// TIA Portal V20 export
FUNCTION_BLOCK "Sequence_1_MainPnP"   // FB246, LAD
AUTHOR : ERsystem_FA2_DH. Kim
// stored: IsIECCheckEnabled true, MemoryReserve 100, Namespace Unit1.Em5, SetENOAutomatically false
   VAR
      instSequenceLADStatus { ExternalWritable := 'False'} : "LAF_StatusLadSequence";
      instSequenceLADControl { ExternalWritable := 'False'} : "LAF_ControlLadSequence";
      statTonTime { ExternalWritable := 'False'} : Array[0..9999] of TON_TIME;
   END_VAR
   VAR_TEMP
      tempCustomerAction : Bool;   // Placeholder for possible actions
      tempDo_nothing_and_wait_for_init : Bool;   // Placeholder for doing nothing
      tempSafeStateCondition : Bool;   // Temp Condition for the equipment module to be in a safe state
   END_VAR
   VAR CONSTANT
      delayTime : Time := T#300ms;
      STEP_IDLE : DInt := 1;
      STEP_IMMEDIATE_STOP : DInt := 9001;   // Step executed when an immediate stop command is triggered for the sequence (i.e. when unit is in state aborting)
      JOB_10_STEP_01 : DInt := 1001;
      JOB_10_STEP_10 : DInt := 1010;
      JOB_10_STEP_11 : DInt := 1011;
      JOB_10_STEP_20 : DInt := 1020;
      JOB_10_STEP_21 : DInt := 1021;
      JOB_10_STEP_22 : DInt := 1022;
      JOB_10_STEP_30 : DInt := 1030;
      JOB_10_STEP_31 : DInt := 1031;
      JOB_10_STEP_40 : DInt := 1040;
      JOB_10_STEP_41 : DInt := 1041;
      JOB_10_STEP_50 : DInt := 1050;
      JOB_10_STEP_60 : DInt := 1060;
      JOB_10_STEP_70 : DInt := 1070;
      JOB_10_STEP_71 : DInt := 1071;
      JOB_10_STEP_80 : DInt := 1080;
      JOB_10_STEP_81 : DInt := 1081;
      JOB_10_STEP_90 : DInt := 1090;
      JOB_1_STEP_01 : DInt := 101;
      JOB_1_STEP_10 : DInt := 110;
      JOB_1_STEP_11 : DInt := 111;
      JOB_1_STEP_12 : DInt := 112;
      JOB_1_STEP_13 : DInt := 113;
      JOB_1_STEP_14 : DInt := 114;
      JOB_1_STEP_15 : DInt := 115;
      JOB_1_STEP_16 : DInt := 116;
      JOB_1_STEP_17 : DInt := 117;
      JOB_1_STEP_18 : DInt := 118;
      JOB_1_STEP_19 : DInt := 119;
      JOB_1_STEP_20 : DInt := 120;
      JOB_1_STEP_21 : DInt := 121;
      JOB_1_STEP_22 : DInt := 122;
      JOB_1_STEP_23 : DInt := 123;
      JOB_1_STEP_24 : DInt := 124;
      JOB_1_STEP_25 : DInt := 125;
      JOB_1_STEP_26 : DInt := 126;
      JOB_1_STEP_27 : DInt := 127;
      JOB_1_STEP_28 : DInt := 128;
      JOB_1_STEP_29 : DInt := 129;
      JOB_1_STEP_30 : DInt := 130;
      JOB_1_STEP_31 : DInt := 131;
      JOB_1_STEP_32 : DInt := 132;
      JOB_1_STEP_33 : DInt := 133;
      JOB_1_STEP_34 : DInt := 134;
      JOB_1_STEP_35 : DInt := 135;
      JOB_1_STEP_36 : DInt := 136;
      JOB_1_STEP_37 : DInt := 137;
      JOB_1_STEP_38 : DInt := 138;
      JOB_1_STEP_39 : DInt := 139;
      JOB_1_STEP_40 : DInt := 140;
      JOB_1_STEP_41 : DInt := 141;
      JOB_1_STEP_42 : DInt := 142;
      JOB_1_STEP_43 : DInt := 143;
      JOB_1_STEP_44 : DInt := 144;
      JOB_1_STEP_45 : DInt := 145;
      JOB_1_STEP_46 : DInt := 146;
      JOB_1_STEP_47 : DInt := 147;
      JOB_1_STEP_48 : DInt := 148;
      JOB_1_STEP_49 : DInt := 149;
      JOB_1_STEP_50 : DInt := 150;
      JOB_1_STEP_80 : DInt := 180;
      JOB_1_STEP_81 : DInt := 181;
      JOB_1_STEP_82 : DInt := 182;
      JOB_1_STEP_83 : DInt := 183;
      JOB_1_STEP_84 : DInt := 184;
      JOB_1_STEP_85 : DInt := 185;
      JOB_1_STEP_86 : DInt := 186;
      JOB_1_STEP_87 : DInt := 187;
      JOB_1_STEP_88 : DInt := 188;
      JOB_1_STEP_89 : DInt := 189;
      JOB_1_STEP_90 : DInt := 190;
      JOB_2_STEP_01 : DInt := 201;
      JOB_2_STEP_10 : DInt := 210;
      JOB_2_STEP_20 : DInt := 220;
      JOB_2_STEP_30 : DInt := 230;
      JOB_2_STEP_40 : DInt := 240;
      JOB_2_STEP_50 : DInt := 250;
      JOB_2_STEP_60 : DInt := 260;
      JOB_2_STEP_80 : DInt := 280;
      JOB_2_STEP_90 : DInt := 290;
      JOB_3_STEP_01 : DInt := 301;
      JOB_3_STEP_10 : DInt := 310;
      JOB_3_STEP_20 : DInt := 320;
      JOB_3_STEP_30 : DInt := 330;
      JOB_3_STEP_40 : DInt := 340;
      JOB_3_STEP_50 : DInt := 350;
      JOB_3_STEP_60 : DInt := 360;
      JOB_3_STEP_80 : DInt := 380;
      JOB_3_STEP_90 : DInt := 390;
      JOB_4_STEP_01 : DInt := 401;
      JOB_4_STEP_20 : DInt := 420;
      JOB_4_STEP_30 : DInt := 430;
      JOB_4_STEP_90 : DInt := 490;
      JOB_5_STEP_01 : DInt := 501;
      JOB_5_STEP_20 : DInt := 520;
      JOB_5_STEP_30 : DInt := 530;
      JOB_5_STEP_40 : DInt := 540;
      JOB_5_STEP_50 : DInt := 550;
      JOB_5_STEP_60 : DInt := 560;
      JOB_5_STEP_80 : DInt := 580;
      JOB_5_STEP_90 : DInt := 590;
      JOB_6_STEP_01 : DInt := 601;
      JOB_6_STEP_10 : DInt := 610;
      JOB_6_STEP_20 : DInt := 620;
      JOB_6_STEP_30 : DInt := 630;
      JOB_6_STEP_40 : DInt := 640;
      JOB_6_STEP_50 : DInt := 650;
      JOB_6_STEP_60 : DInt := 660;
      JOB_6_STEP_80 : DInt := 680;
      JOB_6_STEP_90 : DInt := 690;
      FALSE : Bool := FALSE;
      TRUE : Bool := TRUE;
      kim_bool : Bool := true;
   END_VAR
   VAR_TEMP   // added for the SCL form of the ladder/FBD networks
      _w1 : Bool;
   END_VAR
BEGIN

REGION Network 1: BLOCK INFO HEADER
   // (company) / (C) Copyright (year)
   // ---------------------------------------------------------------------------------
   // Title:                             (Title of this block)
   // Comment/Function: (that is implemented in the block)
   // Library/Family:           (that the source is dedicated to)
   // Author:                        (department / person in charge / contact)
   // Target System:          (test system with FW version)
   // Engineering:              TIA Portal (SW version)
   // Restrictions:               (OB types, etc.)
   // Requirements:           (hardware, technological package, etc.)
   // ---------------------------------------------------------------------------------
   // Change log table:
   // Version          | Date             | Signature      | Expert in charge  | Changes applied ------------------------|----------------------|-------------------------|--------------------------------|-----------------------
   // 001.000.000 | yyyy-mm-dd | 0x00000000 | (name of expert) | First released version
END_REGION

REGION Network 2: DESCRIPTION
   // This is a template block provided by the Automation Framework. It can be used to create an own project.
   // The Block Info Header is prepared to put in your own data.
   // Description of the block could be added here and the docu created by Code2Docu.
END_REGION

REGION Network 3: ********************* CONTROL *************************
END_REGION

REGION Network 4: Sequence Control
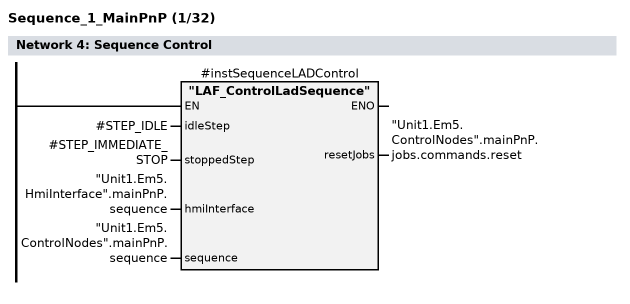
   RUNG wire#powerrail
      #instSequenceLADControl(idleStep := #STEP_IDLE, stoppedStep := #STEP_IMMEDIATE_STOP, hmiInterface := "Unit1.Em5.HmiInterface".mainPnP.sequence, sequence := "Unit1.Em5.ControlNodes".mainPnP.sequence, resetJobs => "Unit1.Em5.ControlNodes".mainPnP.jobs.commands.reset)
   END_RUNG
   // the same network as SCL:
   #instSequenceLADControl(idleStep := #STEP_IDLE,   // "LAF_ControlLadSequence"
                           stoppedStep := #STEP_IMMEDIATE_STOP,
                           hmiInterface := "Unit1.Em5.HmiInterface".mainPnP.sequence,
                           sequence := "Unit1.Em5.ControlNodes".mainPnP.sequence,
                           resetJobs => "Unit1.Em5.ControlNodes".mainPnP.jobs.commands.reset);
END_REGION

REGION Network 5: *************** JOB SELECT **************************
END_REGION

REGION Network 6: STEP IDLE
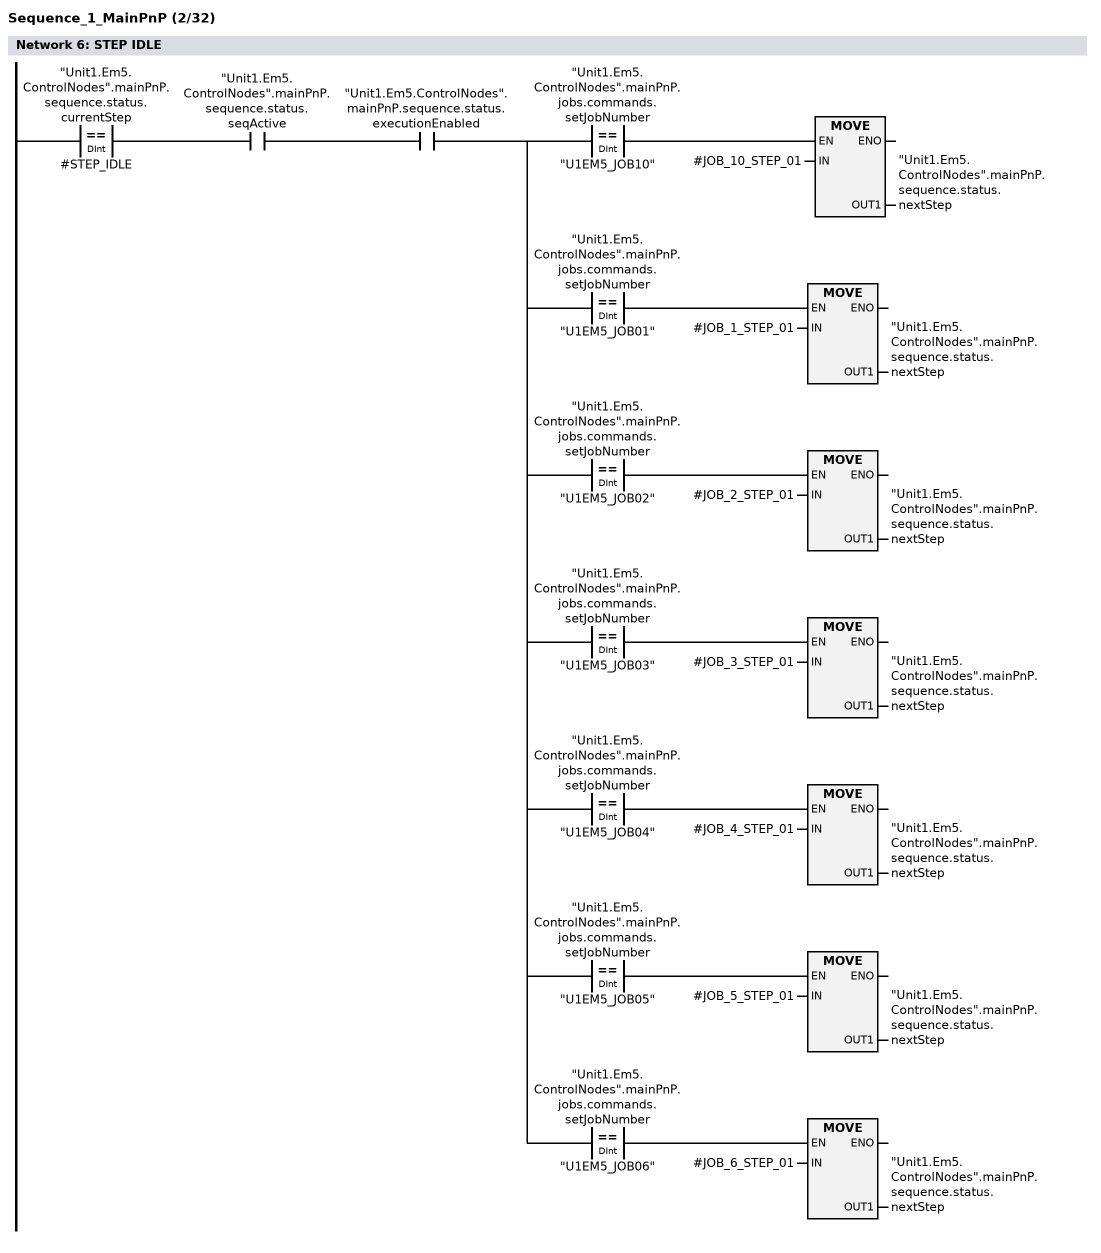
   RUNG wire#powerrail
      { S7_Templates := "SrcType := DInt" } EQ_Contact(in1 := "Unit1.Em5.ControlNodes".mainPnP.sequence.status.currentStep, in2 := #STEP_IDLE)
      Contact( "Unit1.Em5.ControlNodes".mainPnP.sequence.status.seqActive )
      Contact( "Unit1.Em5.ControlNodes".mainPnP.sequence.status.executionEnabled )
      wire#w1
      { S7_Templates := "SrcType := DInt" } EQ_Contact(in1 := "Unit1.Em5.ControlNodes".mainPnP.jobs.commands.setJobNumber, in2 := "U1EM5_JOB10")
      Move(in := #JOB_10_STEP_01, out1 => "Unit1.Em5.ControlNodes".mainPnP.sequence.status.nextStep)
   END_RUNG
   RUNG wire#w1
      { S7_Templates := "SrcType := DInt" } EQ_Contact(in1 := "Unit1.Em5.ControlNodes".mainPnP.jobs.commands.setJobNumber, in2 := "U1EM5_JOB01")
      Move(in := #JOB_1_STEP_01, out1 => "Unit1.Em5.ControlNodes".mainPnP.sequence.status.nextStep)
   END_RUNG
   RUNG wire#w1
      { S7_Templates := "SrcType := DInt" } EQ_Contact(in1 := "Unit1.Em5.ControlNodes".mainPnP.jobs.commands.setJobNumber, in2 := "U1EM5_JOB02")
      Move(in := #JOB_2_STEP_01, out1 => "Unit1.Em5.ControlNodes".mainPnP.sequence.status.nextStep)
   END_RUNG
   RUNG wire#w1
      { S7_Templates := "SrcType := DInt" } EQ_Contact(in1 := "Unit1.Em5.ControlNodes".mainPnP.jobs.commands.setJobNumber, in2 := "U1EM5_JOB03")
      Move(in := #JOB_3_STEP_01, out1 => "Unit1.Em5.ControlNodes".mainPnP.sequence.status.nextStep)
   END_RUNG
   RUNG wire#w1
      { S7_Templates := "SrcType := DInt" } EQ_Contact(in1 := "Unit1.Em5.ControlNodes".mainPnP.jobs.commands.setJobNumber, in2 := "U1EM5_JOB04")
      Move(in := #JOB_4_STEP_01, out1 => "Unit1.Em5.ControlNodes".mainPnP.sequence.status.nextStep)
   END_RUNG
   RUNG wire#w1
      { S7_Templates := "SrcType := DInt" } EQ_Contact(in1 := "Unit1.Em5.ControlNodes".mainPnP.jobs.commands.setJobNumber, in2 := "U1EM5_JOB05")
      Move(in := #JOB_5_STEP_01, out1 => "Unit1.Em5.ControlNodes".mainPnP.sequence.status.nextStep)
   END_RUNG
   RUNG wire#w1
      { S7_Templates := "SrcType := DInt" } EQ_Contact(in1 := "Unit1.Em5.ControlNodes".mainPnP.jobs.commands.setJobNumber, in2 := "U1EM5_JOB06")
      Move(in := #JOB_6_STEP_01, out1 => "Unit1.Em5.ControlNodes".mainPnP.sequence.status.nextStep)
   END_RUNG
   // the same network as SCL:
   #_w1 := ("Unit1.Em5.ControlNodes".mainPnP.sequence.status.currentStep = #STEP_IDLE) AND "Unit1.Em5.ControlNodes".mainPnP.sequence.status.seqActive AND "Unit1.Em5.ControlNodes".mainPnP.sequence.status.executionEnabled;
   IF #_w1 AND ("Unit1.Em5.ControlNodes".mainPnP.jobs.commands.setJobNumber = "U1EM5_JOB10") THEN
       "Unit1.Em5.ControlNodes".mainPnP.sequence.status.nextStep := #JOB_10_STEP_01;
   END_IF;
   IF #_w1 AND ("Unit1.Em5.ControlNodes".mainPnP.jobs.commands.setJobNumber = "U1EM5_JOB01") THEN
       "Unit1.Em5.ControlNodes".mainPnP.sequence.status.nextStep := #JOB_1_STEP_01;
   END_IF;
   IF #_w1 AND ("Unit1.Em5.ControlNodes".mainPnP.jobs.commands.setJobNumber = "U1EM5_JOB02") THEN
       "Unit1.Em5.ControlNodes".mainPnP.sequence.status.nextStep := #JOB_2_STEP_01;
   END_IF;
   IF #_w1 AND ("Unit1.Em5.ControlNodes".mainPnP.jobs.commands.setJobNumber = "U1EM5_JOB03") THEN
       "Unit1.Em5.ControlNodes".mainPnP.sequence.status.nextStep := #JOB_3_STEP_01;
   END_IF;
   IF #_w1 AND ("Unit1.Em5.ControlNodes".mainPnP.jobs.commands.setJobNumber = "U1EM5_JOB04") THEN
       "Unit1.Em5.ControlNodes".mainPnP.sequence.status.nextStep := #JOB_4_STEP_01;
   END_IF;
   IF #_w1 AND ("Unit1.Em5.ControlNodes".mainPnP.jobs.commands.setJobNumber = "U1EM5_JOB05") THEN
       "Unit1.Em5.ControlNodes".mainPnP.sequence.status.nextStep := #JOB_5_STEP_01;
   END_IF;
   IF #_w1 AND ("Unit1.Em5.ControlNodes".mainPnP.jobs.commands.setJobNumber = "U1EM5_JOB06") THEN
       "Unit1.Em5.ControlNodes".mainPnP.sequence.status.nextStep := #JOB_6_STEP_01;
   END_IF;
END_REGION

REGION Network 7: *************** JOB[10] EM HOMING ************************
END_REGION

REGION Network 8: Step[1001] : JOB[10] Condition
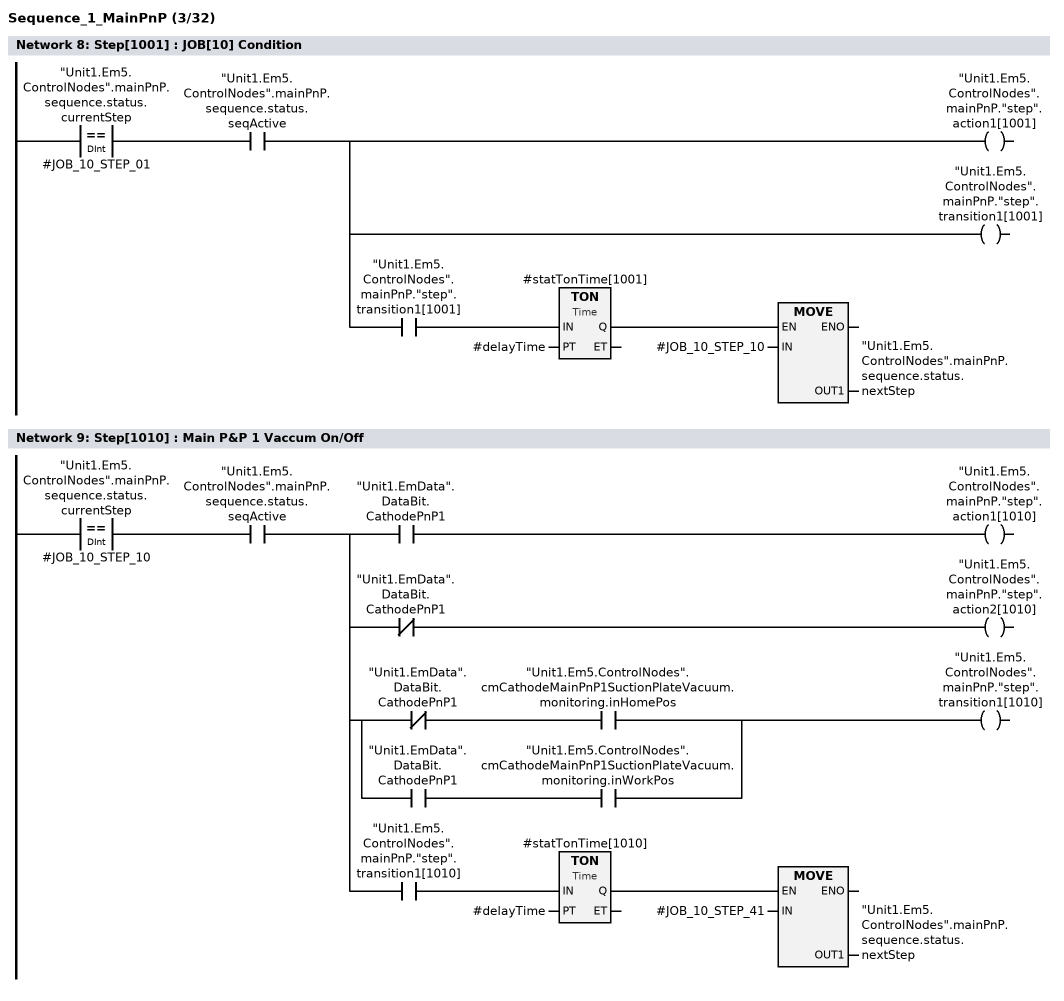
   RUNG wire#powerrail
      { S7_Templates := "SrcType := DInt" } EQ_Contact(in1 := "Unit1.Em5.ControlNodes".mainPnP.sequence.status.currentStep, in2 := #JOB_10_STEP_01)
      Contact( "Unit1.Em5.ControlNodes".mainPnP.sequence.status.seqActive )
      wire#w1
      Coil( "Unit1.Em5.ControlNodes".mainPnP."step".action1[1001] )
   END_RUNG
   RUNG wire#w1
      Coil( "Unit1.Em5.ControlNodes".mainPnP."step".transition1[1001] )
   END_RUNG
   RUNG wire#w1
      Contact( "Unit1.Em5.ControlNodes".mainPnP."step".transition1[1001] )
      { S7_Templates := "time_type := Time" } #statTonTime[1001].TON(pt := #delayTime, et =>)
      Move(in := #JOB_10_STEP_10, out1 => "Unit1.Em5.ControlNodes".mainPnP.sequence.status.nextStep)
   END_RUNG
   // the same network as SCL:
   "Unit1.Em5.ControlNodes".mainPnP."step".action1[1001] := ("Unit1.Em5.ControlNodes".mainPnP.sequence.status.currentStep = #JOB_10_STEP_01) AND "Unit1.Em5.ControlNodes".mainPnP.sequence.status.seqActive;
   "Unit1.Em5.ControlNodes".mainPnP."step".transition1[1001] := ("Unit1.Em5.ControlNodes".mainPnP.sequence.status.currentStep = #JOB_10_STEP_01) AND "Unit1.Em5.ControlNodes".mainPnP.sequence.status.seqActive;
   #statTonTime[1001].TON(IN := ("Unit1.Em5.ControlNodes".mainPnP.sequence.status.currentStep = #JOB_10_STEP_01) AND "Unit1.Em5.ControlNodes".mainPnP.sequence.status.seqActive AND "Unit1.Em5.ControlNodes".mainPnP."step".transition1[1001],
                          PT := #delayTime);
   IF #statTonTime[1001].Q THEN
       "Unit1.Em5.ControlNodes".mainPnP.sequence.status.nextStep := #JOB_10_STEP_10;
   END_IF;
END_REGION

REGION Network 9: Step[1010] : Main P&P 1 Vaccum On/Off
   RUNG wire#powerrail
      { S7_Templates := "SrcType := DInt" } EQ_Contact(in1 := "Unit1.Em5.ControlNodes".mainPnP.sequence.status.currentStep, in2 := #JOB_10_STEP_10)
      Contact( "Unit1.Em5.ControlNodes".mainPnP.sequence.status.seqActive )
      wire#w1
      Contact( "Unit1.EmData".DataBit.CathodePnP1 )
      Coil( "Unit1.Em5.ControlNodes".mainPnP."step".action1[1010] )
   END_RUNG
   RUNG wire#w1
      I_Contact( "Unit1.EmData".DataBit.CathodePnP1 )
      Coil( "Unit1.Em5.ControlNodes".mainPnP."step".action2[1010] )
   END_RUNG
   RUNG wire#w1
      I_Contact( "Unit1.EmData".DataBit.CathodePnP1 )
      Contact( "Unit1.Em5.ControlNodes".cmCathodeMainPnP1SuctionPlateVacuum.monitoring.inHomePos )
      wire#w2
      Coil( "Unit1.Em5.ControlNodes".mainPnP."step".transition1[1010] )
   END_RUNG
   RUNG wire#w1
      Contact( "Unit1.EmData".DataBit.CathodePnP1 )
      Contact( "Unit1.Em5.ControlNodes".cmCathodeMainPnP1SuctionPlateVacuum.monitoring.inWorkPos )
   END_RUNG wire#w2
   RUNG wire#w1
      Contact( "Unit1.Em5.ControlNodes".mainPnP."step".transition1[1010] )
      { S7_Templates := "time_type := Time" } #statTonTime[1010].TON(pt := #delayTime, et =>)
      Move(in := #JOB_10_STEP_41, out1 => "Unit1.Em5.ControlNodes".mainPnP.sequence.status.nextStep)
   END_RUNG
   // the same network as SCL:
   #_w1 := ("Unit1.Em5.ControlNodes".mainPnP.sequence.status.currentStep = #JOB_10_STEP_10) AND "Unit1.Em5.ControlNodes".mainPnP.sequence.status.seqActive;
   "Unit1.Em5.ControlNodes".mainPnP."step".action1[1010] := #_w1 AND "Unit1.EmData".DataBit.CathodePnP1;
   "Unit1.Em5.ControlNodes".mainPnP."step".action2[1010] := #_w1 AND NOT "Unit1.EmData".DataBit.CathodePnP1;
   "Unit1.Em5.ControlNodes".mainPnP."step".transition1[1010] := #_w1 AND ((NOT "Unit1.EmData".DataBit.CathodePnP1 AND "Unit1.Em5.ControlNodes".cmCathodeMainPnP1SuctionPlateVacuum.monitoring.inHomePos) OR ("Unit1.EmData".DataBit.CathodePnP1 AND "Unit1.Em5.ControlNodes".cmCathodeMainPnP1SuctionPlateVacuum.monitoring.inWorkPos));
   #statTonTime[1010].TON(IN := #_w1 AND "Unit1.Em5.ControlNodes".mainPnP."step".transition1[1010],
                          PT := #delayTime);
   IF #statTonTime[1010].Q THEN
       "Unit1.Em5.ControlNodes".mainPnP.sequence.status.nextStep := #JOB_10_STEP_41;
   END_IF;
END_REGION

REGION Network 10: Step[1041] : Main P&P 2 Vaccum On/Off
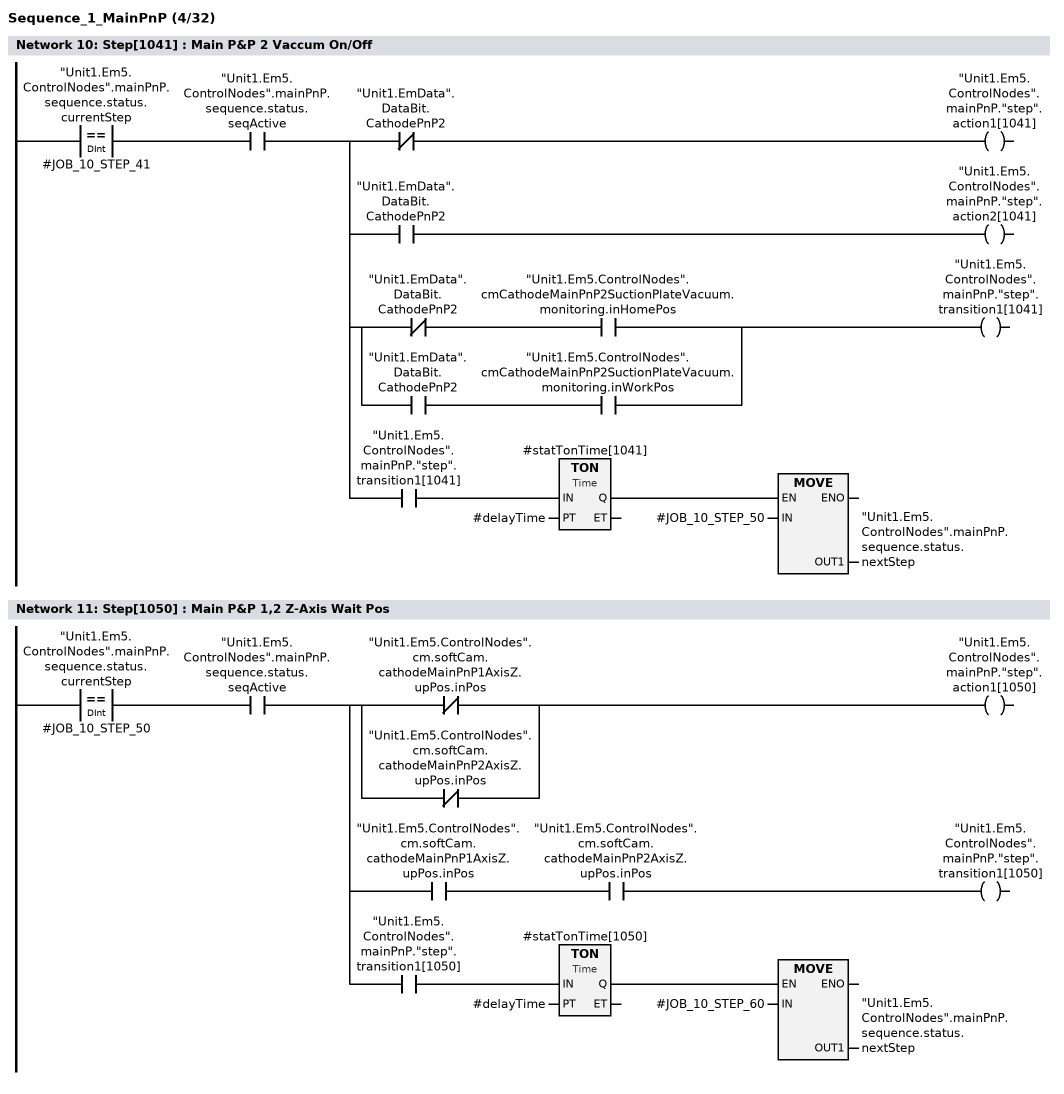
   RUNG wire#powerrail
      { S7_Templates := "SrcType := DInt" } EQ_Contact(in1 := "Unit1.Em5.ControlNodes".mainPnP.sequence.status.currentStep, in2 := #JOB_10_STEP_41)
      Contact( "Unit1.Em5.ControlNodes".mainPnP.sequence.status.seqActive )
      wire#w1
      I_Contact( "Unit1.EmData".DataBit.CathodePnP2 )
      Coil( "Unit1.Em5.ControlNodes".mainPnP."step".action1[1041] )
   END_RUNG
   RUNG wire#w1
      Contact( "Unit1.EmData".DataBit.CathodePnP2 )
      Coil( "Unit1.Em5.ControlNodes".mainPnP."step".action2[1041] )
   END_RUNG
   RUNG wire#w1
      I_Contact( "Unit1.EmData".DataBit.CathodePnP2 )
      Contact( "Unit1.Em5.ControlNodes".cmCathodeMainPnP2SuctionPlateVacuum.monitoring.inHomePos )
      wire#w2
      Coil( "Unit1.Em5.ControlNodes".mainPnP."step".transition1[1041] )
   END_RUNG
   RUNG wire#w1
      Contact( "Unit1.EmData".DataBit.CathodePnP2 )
      Contact( "Unit1.Em5.ControlNodes".cmCathodeMainPnP2SuctionPlateVacuum.monitoring.inWorkPos )
   END_RUNG wire#w2
   RUNG wire#w1
      Contact( "Unit1.Em5.ControlNodes".mainPnP."step".transition1[1041] )
      { S7_Templates := "time_type := Time" } #statTonTime[1041].TON(pt := #delayTime, et =>)
      Move(in := #JOB_10_STEP_50, out1 => "Unit1.Em5.ControlNodes".mainPnP.sequence.status.nextStep)
   END_RUNG
   // the same network as SCL:
   #_w1 := ("Unit1.Em5.ControlNodes".mainPnP.sequence.status.currentStep = #JOB_10_STEP_41) AND "Unit1.Em5.ControlNodes".mainPnP.sequence.status.seqActive;
   "Unit1.Em5.ControlNodes".mainPnP."step".action1[1041] := #_w1 AND NOT "Unit1.EmData".DataBit.CathodePnP2;
   "Unit1.Em5.ControlNodes".mainPnP."step".action2[1041] := #_w1 AND "Unit1.EmData".DataBit.CathodePnP2;
   "Unit1.Em5.ControlNodes".mainPnP."step".transition1[1041] := #_w1 AND ((NOT "Unit1.EmData".DataBit.CathodePnP2 AND "Unit1.Em5.ControlNodes".cmCathodeMainPnP2SuctionPlateVacuum.monitoring.inHomePos) OR ("Unit1.EmData".DataBit.CathodePnP2 AND "Unit1.Em5.ControlNodes".cmCathodeMainPnP2SuctionPlateVacuum.monitoring.inWorkPos));
   #statTonTime[1041].TON(IN := #_w1 AND "Unit1.Em5.ControlNodes".mainPnP."step".transition1[1041],
                          PT := #delayTime);
   IF #statTonTime[1041].Q THEN
       "Unit1.Em5.ControlNodes".mainPnP.sequence.status.nextStep := #JOB_10_STEP_50;
   END_IF;
END_REGION

REGION Network 11: Step[1050] : Main P&P 1,2 Z-Axis Wait Pos
   RUNG wire#powerrail
      { S7_Templates := "SrcType := DInt" } EQ_Contact(in1 := "Unit1.Em5.ControlNodes".mainPnP.sequence.status.currentStep, in2 := #JOB_10_STEP_50)
      Contact( "Unit1.Em5.ControlNodes".mainPnP.sequence.status.seqActive )
      wire#w1
      I_Contact( "Unit1.Em5.ControlNodes".cm.softCam.cathodeMainPnP1AxisZ.upPos.inPos )
      wire#w2
      Coil( "Unit1.Em5.ControlNodes".mainPnP."step".action1[1050] )
   END_RUNG
   RUNG wire#w1
      I_Contact( "Unit1.Em5.ControlNodes".cm.softCam.cathodeMainPnP2AxisZ.upPos.inPos )
   END_RUNG wire#w2
   RUNG wire#w1
      Contact( "Unit1.Em5.ControlNodes".cm.softCam.cathodeMainPnP1AxisZ.upPos.inPos )
      Contact( "Unit1.Em5.ControlNodes".cm.softCam.cathodeMainPnP2AxisZ.upPos.inPos )
      Coil( "Unit1.Em5.ControlNodes".mainPnP."step".transition1[1050] )
   END_RUNG
   RUNG wire#w1
      Contact( "Unit1.Em5.ControlNodes".mainPnP."step".transition1[1050] )
      { S7_Templates := "time_type := Time" } #statTonTime[1050].TON(pt := #delayTime, et =>)
      Move(in := #JOB_10_STEP_60, out1 => "Unit1.Em5.ControlNodes".mainPnP.sequence.status.nextStep)
   END_RUNG
   // the same network as SCL:
   #_w1 := ("Unit1.Em5.ControlNodes".mainPnP.sequence.status.currentStep = #JOB_10_STEP_50) AND "Unit1.Em5.ControlNodes".mainPnP.sequence.status.seqActive;
   "Unit1.Em5.ControlNodes".mainPnP."step".action1[1050] := #_w1 AND (NOT "Unit1.Em5.ControlNodes".cm.softCam.cathodeMainPnP1AxisZ.upPos.inPos OR NOT "Unit1.Em5.ControlNodes".cm.softCam.cathodeMainPnP2AxisZ.upPos.inPos);
   "Unit1.Em5.ControlNodes".mainPnP."step".transition1[1050] := #_w1 AND "Unit1.Em5.ControlNodes".cm.softCam.cathodeMainPnP1AxisZ.upPos.inPos AND "Unit1.Em5.ControlNodes".cm.softCam.cathodeMainPnP2AxisZ.upPos.inPos;
   #statTonTime[1050].TON(IN := #_w1 AND "Unit1.Em5.ControlNodes".mainPnP."step".transition1[1050],
                          PT := #delayTime);
   IF #statTonTime[1050].Q THEN
       "Unit1.Em5.ControlNodes".mainPnP.sequence.status.nextStep := #JOB_10_STEP_60;
   END_IF;
END_REGION

REGION Network 12: Step[1060] : Main P&P 1 Y-Axis Wait Pos
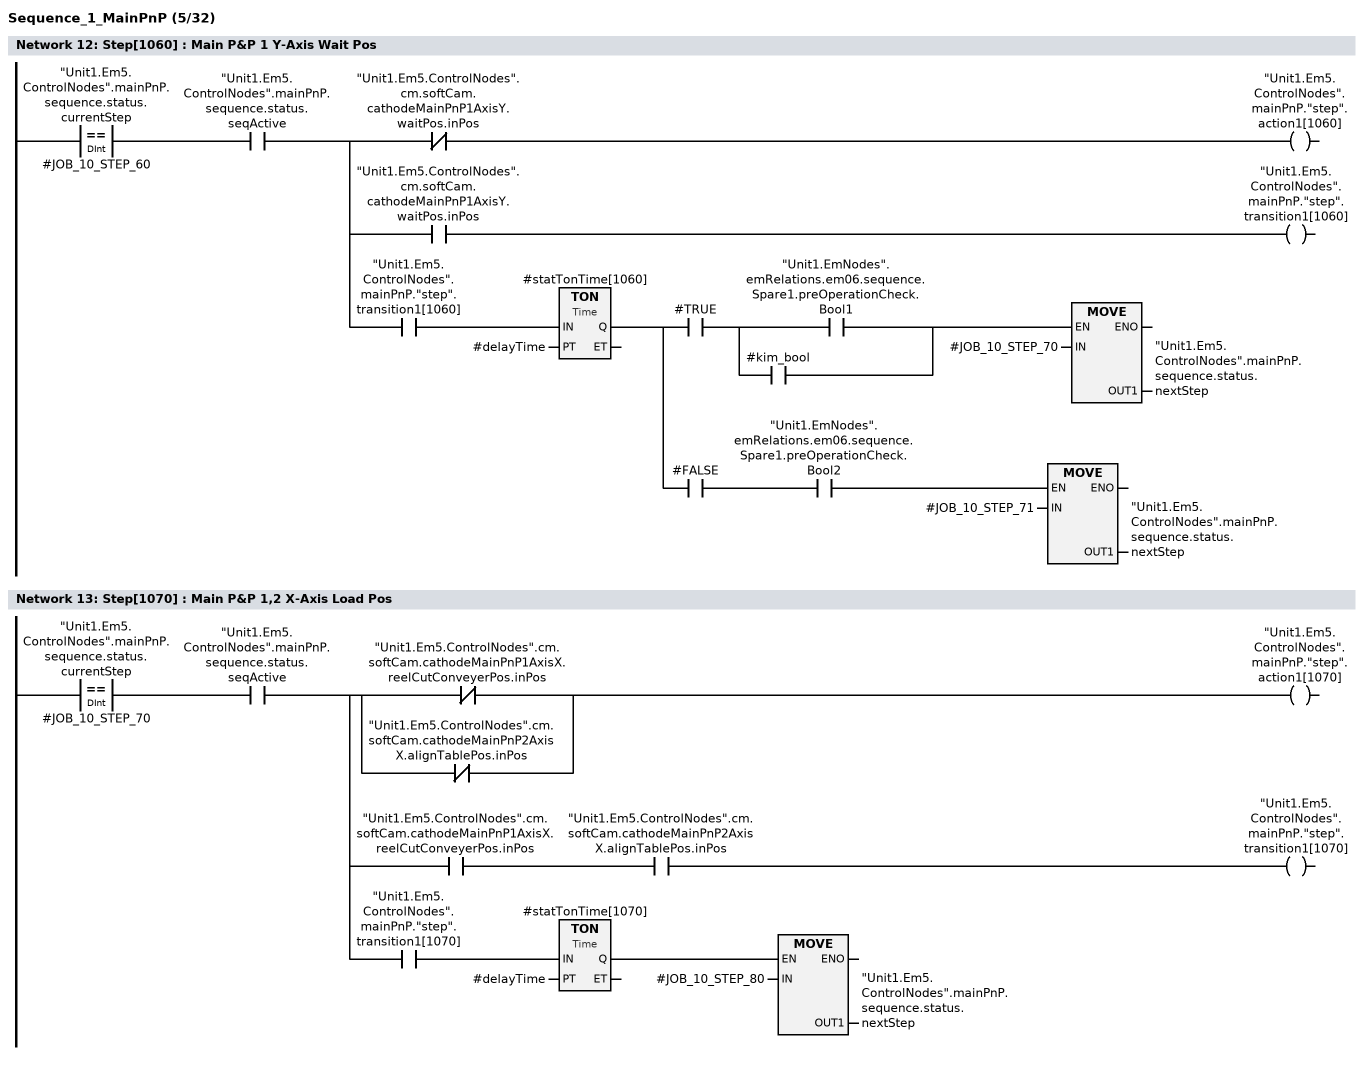
   RUNG wire#powerrail
      { S7_Templates := "SrcType := DInt" } EQ_Contact(in1 := "Unit1.Em5.ControlNodes".mainPnP.sequence.status.currentStep, in2 := #JOB_10_STEP_60)
      Contact( "Unit1.Em5.ControlNodes".mainPnP.sequence.status.seqActive )
      wire#w1
      I_Contact( "Unit1.Em5.ControlNodes".cm.softCam.cathodeMainPnP1AxisY.waitPos.inPos )
      Coil( "Unit1.Em5.ControlNodes".mainPnP."step".action1[1060] )
   END_RUNG
   RUNG wire#w1
      Contact( "Unit1.Em5.ControlNodes".cm.softCam.cathodeMainPnP1AxisY.waitPos.inPos )
      Coil( "Unit1.Em5.ControlNodes".mainPnP."step".transition1[1060] )
   END_RUNG
   RUNG wire#w1
      Contact( "Unit1.Em5.ControlNodes".mainPnP."step".transition1[1060] )
      { S7_Templates := "time_type := Time" } #statTonTime[1060].TON(pt := #delayTime, et =>)
      wire#w2
      Contact( #TRUE )
      wire#w3
      Contact( "Unit1.EmNodes".emRelations.em06.sequence.Spare1.preOperationCheck.Bool1 )
      wire#w4
      Move(in := #JOB_10_STEP_70, out1 => "Unit1.Em5.ControlNodes".mainPnP.sequence.status.nextStep)
   END_RUNG
   RUNG wire#w3
      Contact( #kim_bool )
   END_RUNG wire#w4
   RUNG wire#w2
      Contact( #FALSE )
      Contact( "Unit1.EmNodes".emRelations.em06.sequence.Spare1.preOperationCheck.Bool2 )
      Move(in := #JOB_10_STEP_71, out1 => "Unit1.Em5.ControlNodes".mainPnP.sequence.status.nextStep)
   END_RUNG
   // the same network as SCL:
   #_w1 := ("Unit1.Em5.ControlNodes".mainPnP.sequence.status.currentStep = #JOB_10_STEP_60) AND "Unit1.Em5.ControlNodes".mainPnP.sequence.status.seqActive;
   "Unit1.Em5.ControlNodes".mainPnP."step".action1[1060] := #_w1 AND NOT "Unit1.Em5.ControlNodes".cm.softCam.cathodeMainPnP1AxisY.waitPos.inPos;
   "Unit1.Em5.ControlNodes".mainPnP."step".transition1[1060] := #_w1 AND "Unit1.Em5.ControlNodes".cm.softCam.cathodeMainPnP1AxisY.waitPos.inPos;
   #statTonTime[1060].TON(IN := #_w1 AND "Unit1.Em5.ControlNodes".mainPnP."step".transition1[1060],
                          PT := #delayTime);
   IF #statTonTime[1060].Q AND #TRUE AND ("Unit1.EmNodes".emRelations.em06.sequence.Spare1.preOperationCheck.Bool1 OR #kim_bool) THEN
       "Unit1.Em5.ControlNodes".mainPnP.sequence.status.nextStep := #JOB_10_STEP_70;
   END_IF;
   IF #statTonTime[1060].Q AND #FALSE AND "Unit1.EmNodes".emRelations.em06.sequence.Spare1.preOperationCheck.Bool2 THEN
       "Unit1.Em5.ControlNodes".mainPnP.sequence.status.nextStep := #JOB_10_STEP_71;
   END_IF;
END_REGION

REGION Network 13: Step[1070] : Main P&P 1,2 X-Axis Load Pos
   RUNG wire#powerrail
      { S7_Templates := "SrcType := DInt" } EQ_Contact(in1 := "Unit1.Em5.ControlNodes".mainPnP.sequence.status.currentStep, in2 := #JOB_10_STEP_70)
      Contact( "Unit1.Em5.ControlNodes".mainPnP.sequence.status.seqActive )
      wire#w1
      I_Contact( "Unit1.Em5.ControlNodes".cm.softCam.cathodeMainPnP1AxisX.reelCutConveyerPos.inPos )
      wire#w2
      Coil( "Unit1.Em5.ControlNodes".mainPnP."step".action1[1070] )
   END_RUNG
   RUNG wire#w1
      I_Contact( "Unit1.Em5.ControlNodes".cm.softCam.cathodeMainPnP2AxisX.alignTablePos.inPos )
   END_RUNG wire#w2
   RUNG wire#w1
      Contact( "Unit1.Em5.ControlNodes".cm.softCam.cathodeMainPnP1AxisX.reelCutConveyerPos.inPos )
      Contact( "Unit1.Em5.ControlNodes".cm.softCam.cathodeMainPnP2AxisX.alignTablePos.inPos )
      Coil( "Unit1.Em5.ControlNodes".mainPnP."step".transition1[1070] )
   END_RUNG
   RUNG wire#w1
      Contact( "Unit1.Em5.ControlNodes".mainPnP."step".transition1[1070] )
      { S7_Templates := "time_type := Time" } #statTonTime[1070].TON(pt := #delayTime, et =>)
      Move(in := #JOB_10_STEP_80, out1 => "Unit1.Em5.ControlNodes".mainPnP.sequence.status.nextStep)
   END_RUNG
   // the same network as SCL:
   #_w1 := ("Unit1.Em5.ControlNodes".mainPnP.sequence.status.currentStep = #JOB_10_STEP_70) AND "Unit1.Em5.ControlNodes".mainPnP.sequence.status.seqActive;
   "Unit1.Em5.ControlNodes".mainPnP."step".action1[1070] := #_w1 AND (NOT "Unit1.Em5.ControlNodes".cm.softCam.cathodeMainPnP1AxisX.reelCutConveyerPos.inPos OR NOT "Unit1.Em5.ControlNodes".cm.softCam.cathodeMainPnP2AxisX.alignTablePos.inPos);
   "Unit1.Em5.ControlNodes".mainPnP."step".transition1[1070] := #_w1 AND "Unit1.Em5.ControlNodes".cm.softCam.cathodeMainPnP1AxisX.reelCutConveyerPos.inPos AND "Unit1.Em5.ControlNodes".cm.softCam.cathodeMainPnP2AxisX.alignTablePos.inPos;
   #statTonTime[1070].TON(IN := #_w1 AND "Unit1.Em5.ControlNodes".mainPnP."step".transition1[1070],
                          PT := #delayTime);
   IF #statTonTime[1070].Q THEN
       "Unit1.Em5.ControlNodes".mainPnP.sequence.status.nextStep := #JOB_10_STEP_80;
   END_IF;
END_REGION

REGION Network 14: Step[1080] : Main P&P 1 Rotary Cylinder InHomePos
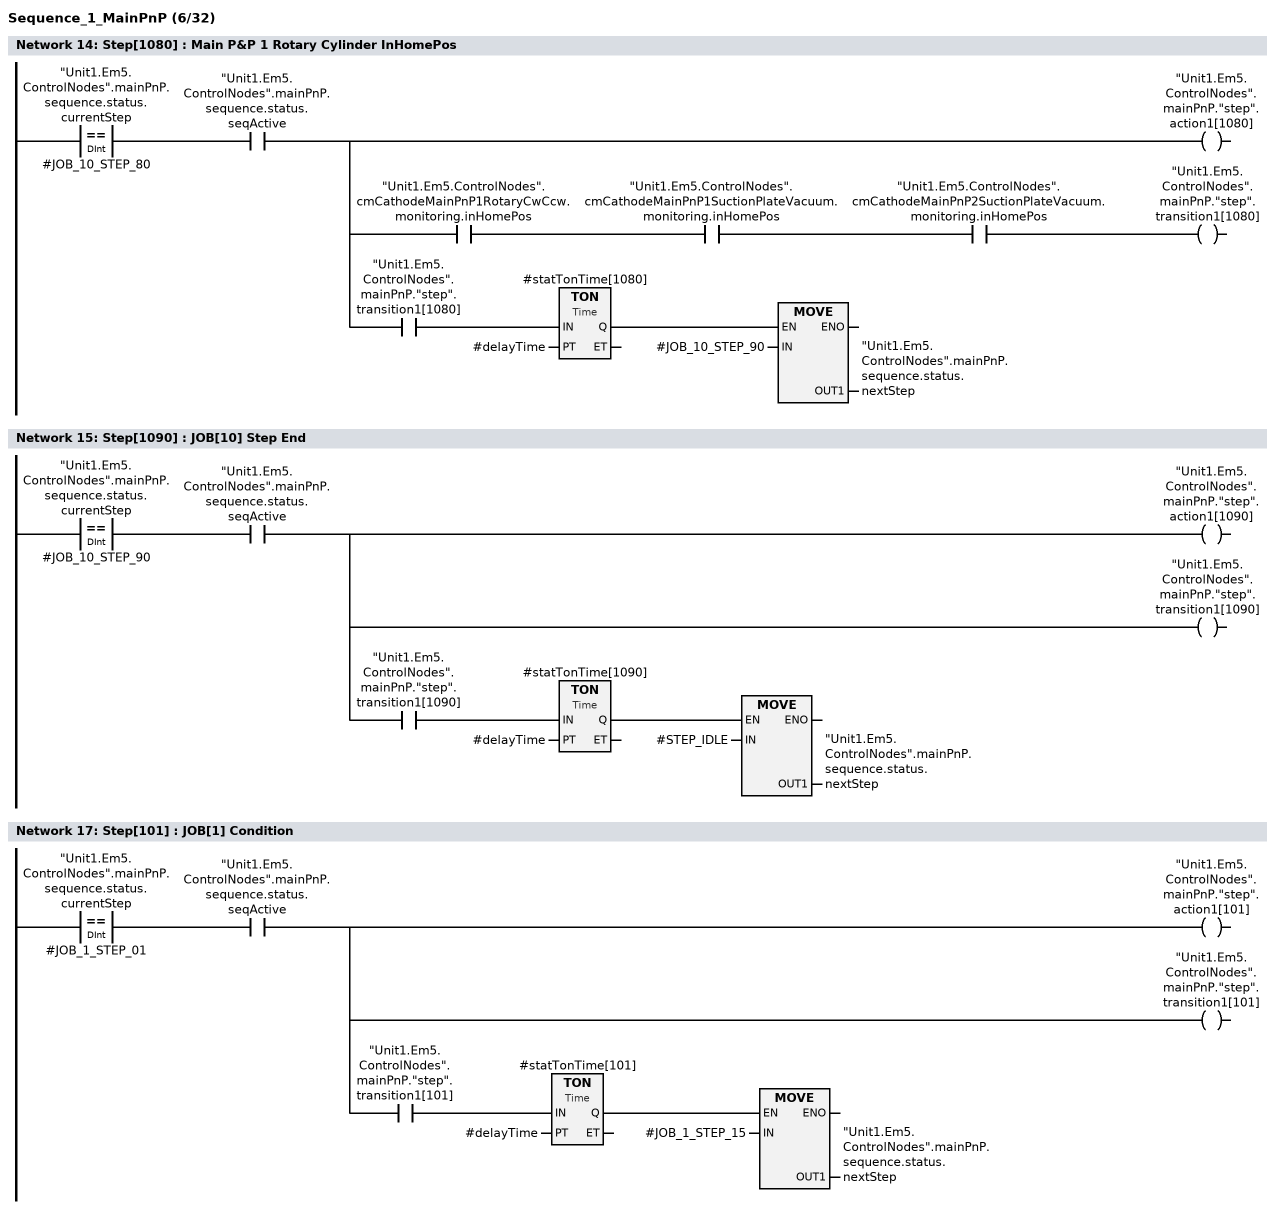
   RUNG wire#powerrail
      { S7_Templates := "SrcType := DInt" } EQ_Contact(in1 := "Unit1.Em5.ControlNodes".mainPnP.sequence.status.currentStep, in2 := #JOB_10_STEP_80)
      Contact( "Unit1.Em5.ControlNodes".mainPnP.sequence.status.seqActive )
      wire#w1
      Coil( "Unit1.Em5.ControlNodes".mainPnP."step".action1[1080] )
   END_RUNG
   RUNG wire#w1
      Contact( "Unit1.Em5.ControlNodes".cmCathodeMainPnP1RotaryCwCcw.monitoring.inHomePos )
      Contact( "Unit1.Em5.ControlNodes".cmCathodeMainPnP1SuctionPlateVacuum.monitoring.inHomePos )
      Contact( "Unit1.Em5.ControlNodes".cmCathodeMainPnP2SuctionPlateVacuum.monitoring.inHomePos )
      Coil( "Unit1.Em5.ControlNodes".mainPnP."step".transition1[1080] )
   END_RUNG
   RUNG wire#w1
      Contact( "Unit1.Em5.ControlNodes".mainPnP."step".transition1[1080] )
      { S7_Templates := "time_type := Time" } #statTonTime[1080].TON(pt := #delayTime, et =>)
      Move(in := #JOB_10_STEP_90, out1 => "Unit1.Em5.ControlNodes".mainPnP.sequence.status.nextStep)
   END_RUNG
   // the same network as SCL:
   "Unit1.Em5.ControlNodes".mainPnP."step".action1[1080] := ("Unit1.Em5.ControlNodes".mainPnP.sequence.status.currentStep = #JOB_10_STEP_80) AND "Unit1.Em5.ControlNodes".mainPnP.sequence.status.seqActive;
   "Unit1.Em5.ControlNodes".mainPnP."step".transition1[1080] := ("Unit1.Em5.ControlNodes".mainPnP.sequence.status.currentStep = #JOB_10_STEP_80) AND "Unit1.Em5.ControlNodes".mainPnP.sequence.status.seqActive AND "Unit1.Em5.ControlNodes".cmCathodeMainPnP1RotaryCwCcw.monitoring.inHomePos AND "Unit1.Em5.ControlNodes".cmCathodeMainPnP1SuctionPlateVacuum.monitoring.inHomePos AND "Unit1.Em5.ControlNodes".cmCathodeMainPnP2SuctionPlateVacuum.monitoring.inHomePos;
   #statTonTime[1080].TON(IN := ("Unit1.Em5.ControlNodes".mainPnP.sequence.status.currentStep = #JOB_10_STEP_80) AND "Unit1.Em5.ControlNodes".mainPnP.sequence.status.seqActive AND "Unit1.Em5.ControlNodes".mainPnP."step".transition1[1080],
                          PT := #delayTime);
   IF #statTonTime[1080].Q THEN
       "Unit1.Em5.ControlNodes".mainPnP.sequence.status.nextStep := #JOB_10_STEP_90;
   END_IF;
END_REGION

REGION Network 15: Step[1090] : JOB[10] Step End
   RUNG wire#powerrail
      { S7_Templates := "SrcType := DInt" } EQ_Contact(in1 := "Unit1.Em5.ControlNodes".mainPnP.sequence.status.currentStep, in2 := #JOB_10_STEP_90)
      Contact( "Unit1.Em5.ControlNodes".mainPnP.sequence.status.seqActive )
      wire#w1
      Coil( "Unit1.Em5.ControlNodes".mainPnP."step".action1[1090] )
   END_RUNG
   RUNG wire#w1
      Coil( "Unit1.Em5.ControlNodes".mainPnP."step".transition1[1090] )
   END_RUNG
   RUNG wire#w1
      Contact( "Unit1.Em5.ControlNodes".mainPnP."step".transition1[1090] )
      { S7_Templates := "time_type := Time" } #statTonTime[1090].TON(pt := #delayTime, et =>)
      Move(in := #STEP_IDLE, out1 => "Unit1.Em5.ControlNodes".mainPnP.sequence.status.nextStep)
   END_RUNG
   // the same network as SCL:
   "Unit1.Em5.ControlNodes".mainPnP."step".action1[1090] := ("Unit1.Em5.ControlNodes".mainPnP.sequence.status.currentStep = #JOB_10_STEP_90) AND "Unit1.Em5.ControlNodes".mainPnP.sequence.status.seqActive;
   "Unit1.Em5.ControlNodes".mainPnP."step".transition1[1090] := ("Unit1.Em5.ControlNodes".mainPnP.sequence.status.currentStep = #JOB_10_STEP_90) AND "Unit1.Em5.ControlNodes".mainPnP.sequence.status.seqActive;
   #statTonTime[1090].TON(IN := ("Unit1.Em5.ControlNodes".mainPnP.sequence.status.currentStep = #JOB_10_STEP_90) AND "Unit1.Em5.ControlNodes".mainPnP.sequence.status.seqActive AND "Unit1.Em5.ControlNodes".mainPnP."step".transition1[1090],
                          PT := #delayTime);
   IF #statTonTime[1090].Q THEN
       "Unit1.Em5.ControlNodes".mainPnP.sequence.status.nextStep := #STEP_IDLE;
   END_IF;
END_REGION

REGION Network 16: *************** JOB[1] EM HOMING ************************
END_REGION

REGION Network 17: Step[101] : JOB[1] Condition
   RUNG wire#powerrail
      { S7_Templates := "SrcType := DInt" } EQ_Contact(in1 := "Unit1.Em5.ControlNodes".mainPnP.sequence.status.currentStep, in2 := #JOB_1_STEP_01)
      Contact( "Unit1.Em5.ControlNodes".mainPnP.sequence.status.seqActive )
      wire#w1
      Coil( "Unit1.Em5.ControlNodes".mainPnP."step".action1[101] )
   END_RUNG
   RUNG wire#w1
      Coil( "Unit1.Em5.ControlNodes".mainPnP."step".transition1[101] )
   END_RUNG
   RUNG wire#w1
      Contact( "Unit1.Em5.ControlNodes".mainPnP."step".transition1[101] )
      { S7_Templates := "time_type := Time" } #statTonTime[101].TON(pt := #delayTime, et =>)
      Move(in := #JOB_1_STEP_15, out1 => "Unit1.Em5.ControlNodes".mainPnP.sequence.status.nextStep)
   END_RUNG
   // the same network as SCL:
   "Unit1.Em5.ControlNodes".mainPnP."step".action1[101] := ("Unit1.Em5.ControlNodes".mainPnP.sequence.status.currentStep = #JOB_1_STEP_01) AND "Unit1.Em5.ControlNodes".mainPnP.sequence.status.seqActive;
   "Unit1.Em5.ControlNodes".mainPnP."step".transition1[101] := ("Unit1.Em5.ControlNodes".mainPnP.sequence.status.currentStep = #JOB_1_STEP_01) AND "Unit1.Em5.ControlNodes".mainPnP.sequence.status.seqActive;
   #statTonTime[101].TON(IN := ("Unit1.Em5.ControlNodes".mainPnP.sequence.status.currentStep = #JOB_1_STEP_01) AND "Unit1.Em5.ControlNodes".mainPnP.sequence.status.seqActive AND "Unit1.Em5.ControlNodes".mainPnP."step".transition1[101],
                         PT := #delayTime);
   IF #statTonTime[101].Q THEN
       "Unit1.Em5.ControlNodes".mainPnP.sequence.status.nextStep := #JOB_1_STEP_15;
   END_IF;
END_REGION

REGION Network 18: Step[110] : Main P&P 1 Z-Axis Wait Pos
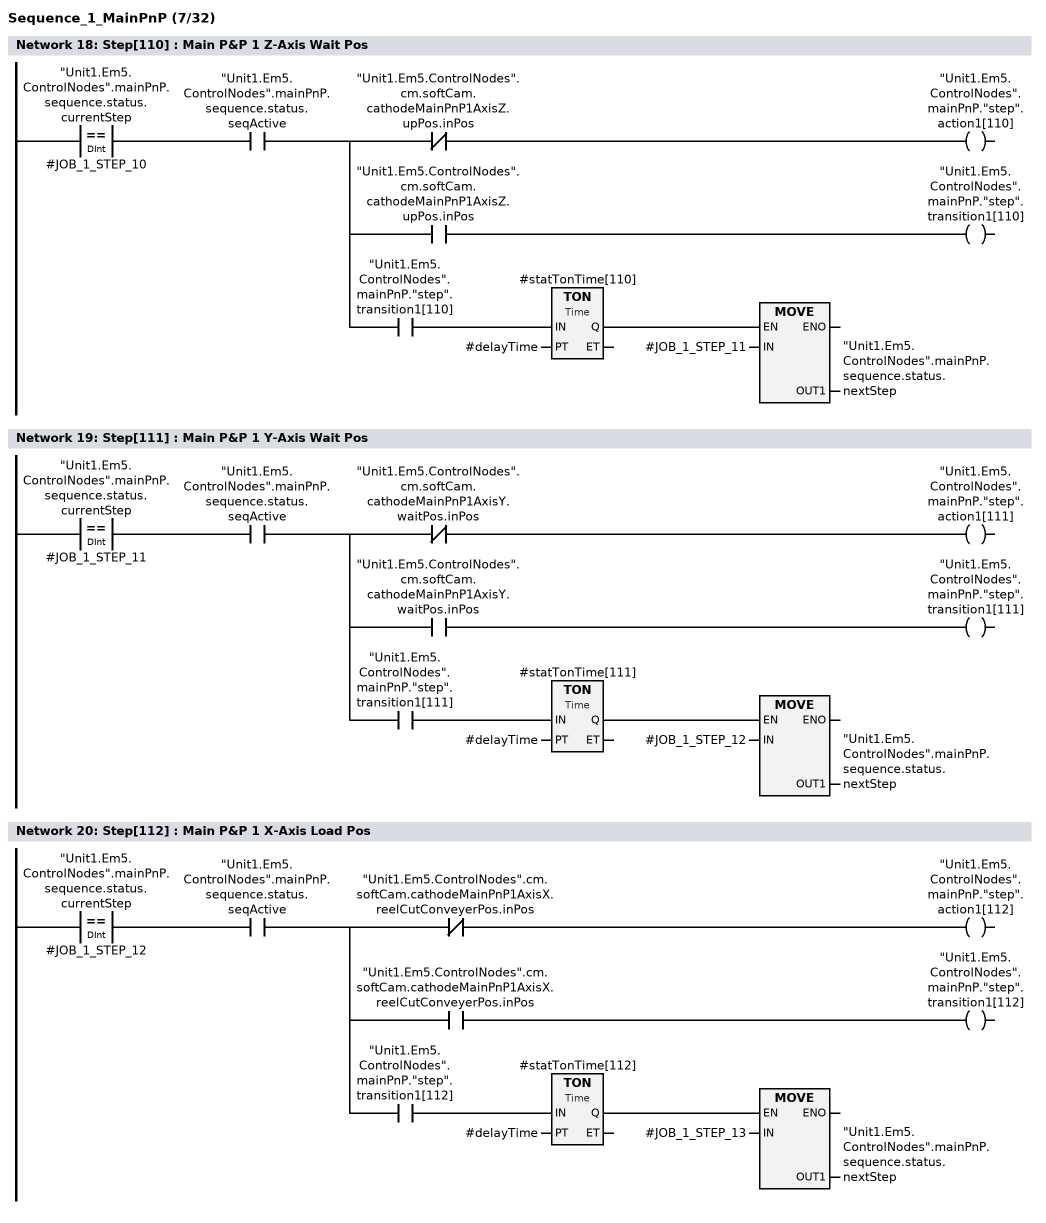
   RUNG wire#powerrail
      { S7_Templates := "SrcType := DInt" } EQ_Contact(in1 := "Unit1.Em5.ControlNodes".mainPnP.sequence.status.currentStep, in2 := #JOB_1_STEP_10)
      Contact( "Unit1.Em5.ControlNodes".mainPnP.sequence.status.seqActive )
      wire#w1
      I_Contact( "Unit1.Em5.ControlNodes".cm.softCam.cathodeMainPnP1AxisZ.upPos.inPos )
      Coil( "Unit1.Em5.ControlNodes".mainPnP."step".action1[110] )
   END_RUNG
   RUNG wire#w1
      Contact( "Unit1.Em5.ControlNodes".cm.softCam.cathodeMainPnP1AxisZ.upPos.inPos )
      Coil( "Unit1.Em5.ControlNodes".mainPnP."step".transition1[110] )
   END_RUNG
   RUNG wire#w1
      Contact( "Unit1.Em5.ControlNodes".mainPnP."step".transition1[110] )
      { S7_Templates := "time_type := Time" } #statTonTime[110].TON(pt := #delayTime, et =>)
      Move(in := #JOB_1_STEP_11, out1 => "Unit1.Em5.ControlNodes".mainPnP.sequence.status.nextStep)
   END_RUNG
   // the same network as SCL:
   #_w1 := ("Unit1.Em5.ControlNodes".mainPnP.sequence.status.currentStep = #JOB_1_STEP_10) AND "Unit1.Em5.ControlNodes".mainPnP.sequence.status.seqActive;
   "Unit1.Em5.ControlNodes".mainPnP."step".action1[110] := #_w1 AND NOT "Unit1.Em5.ControlNodes".cm.softCam.cathodeMainPnP1AxisZ.upPos.inPos;
   "Unit1.Em5.ControlNodes".mainPnP."step".transition1[110] := #_w1 AND "Unit1.Em5.ControlNodes".cm.softCam.cathodeMainPnP1AxisZ.upPos.inPos;
   #statTonTime[110].TON(IN := #_w1 AND "Unit1.Em5.ControlNodes".mainPnP."step".transition1[110],
                         PT := #delayTime);
   IF #statTonTime[110].Q THEN
       "Unit1.Em5.ControlNodes".mainPnP.sequence.status.nextStep := #JOB_1_STEP_11;
   END_IF;
END_REGION

REGION Network 19: Step[111] : Main P&P 1 Y-Axis Wait Pos
   RUNG wire#powerrail
      { S7_Templates := "SrcType := DInt" } EQ_Contact(in1 := "Unit1.Em5.ControlNodes".mainPnP.sequence.status.currentStep, in2 := #JOB_1_STEP_11)
      Contact( "Unit1.Em5.ControlNodes".mainPnP.sequence.status.seqActive )
      wire#w1
      I_Contact( "Unit1.Em5.ControlNodes".cm.softCam.cathodeMainPnP1AxisY.waitPos.inPos )
      Coil( "Unit1.Em5.ControlNodes".mainPnP."step".action1[111] )
   END_RUNG
   RUNG wire#w1
      Contact( "Unit1.Em5.ControlNodes".cm.softCam.cathodeMainPnP1AxisY.waitPos.inPos )
      Coil( "Unit1.Em5.ControlNodes".mainPnP."step".transition1[111] )
   END_RUNG
   RUNG wire#w1
      Contact( "Unit1.Em5.ControlNodes".mainPnP."step".transition1[111] )
      { S7_Templates := "time_type := Time" } #statTonTime[111].TON(pt := #delayTime, et =>)
      Move(in := #JOB_1_STEP_12, out1 => "Unit1.Em5.ControlNodes".mainPnP.sequence.status.nextStep)
   END_RUNG
   // the same network as SCL:
   #_w1 := ("Unit1.Em5.ControlNodes".mainPnP.sequence.status.currentStep = #JOB_1_STEP_11) AND "Unit1.Em5.ControlNodes".mainPnP.sequence.status.seqActive;
   "Unit1.Em5.ControlNodes".mainPnP."step".action1[111] := #_w1 AND NOT "Unit1.Em5.ControlNodes".cm.softCam.cathodeMainPnP1AxisY.waitPos.inPos;
   "Unit1.Em5.ControlNodes".mainPnP."step".transition1[111] := #_w1 AND "Unit1.Em5.ControlNodes".cm.softCam.cathodeMainPnP1AxisY.waitPos.inPos;
   #statTonTime[111].TON(IN := #_w1 AND "Unit1.Em5.ControlNodes".mainPnP."step".transition1[111],
                         PT := #delayTime);
   IF #statTonTime[111].Q THEN
       "Unit1.Em5.ControlNodes".mainPnP.sequence.status.nextStep := #JOB_1_STEP_12;
   END_IF;
END_REGION

REGION Network 20: Step[112] : Main P&P 1 X-Axis Load Pos
   RUNG wire#powerrail
      { S7_Templates := "SrcType := DInt" } EQ_Contact(in1 := "Unit1.Em5.ControlNodes".mainPnP.sequence.status.currentStep, in2 := #JOB_1_STEP_12)
      Contact( "Unit1.Em5.ControlNodes".mainPnP.sequence.status.seqActive )
      wire#w1
      I_Contact( "Unit1.Em5.ControlNodes".cm.softCam.cathodeMainPnP1AxisX.reelCutConveyerPos.inPos )
      Coil( "Unit1.Em5.ControlNodes".mainPnP."step".action1[112] )
   END_RUNG
   RUNG wire#w1
      Contact( "Unit1.Em5.ControlNodes".cm.softCam.cathodeMainPnP1AxisX.reelCutConveyerPos.inPos )
      Coil( "Unit1.Em5.ControlNodes".mainPnP."step".transition1[112] )
   END_RUNG
   RUNG wire#w1
      Contact( "Unit1.Em5.ControlNodes".mainPnP."step".transition1[112] )
      { S7_Templates := "time_type := Time" } #statTonTime[112].TON(pt := #delayTime, et =>)
      Move(in := #JOB_1_STEP_13, out1 => "Unit1.Em5.ControlNodes".mainPnP.sequence.status.nextStep)
   END_RUNG
   // the same network as SCL:
   #_w1 := ("Unit1.Em5.ControlNodes".mainPnP.sequence.status.currentStep = #JOB_1_STEP_12) AND "Unit1.Em5.ControlNodes".mainPnP.sequence.status.seqActive;
   "Unit1.Em5.ControlNodes".mainPnP."step".action1[112] := #_w1 AND NOT "Unit1.Em5.ControlNodes".cm.softCam.cathodeMainPnP1AxisX.reelCutConveyerPos.inPos;
   "Unit1.Em5.ControlNodes".mainPnP."step".transition1[112] := #_w1 AND "Unit1.Em5.ControlNodes".cm.softCam.cathodeMainPnP1AxisX.reelCutConveyerPos.inPos;
   #statTonTime[112].TON(IN := #_w1 AND "Unit1.Em5.ControlNodes".mainPnP."step".transition1[112],
                         PT := #delayTime);
   IF #statTonTime[112].Q THEN
       "Unit1.Em5.ControlNodes".mainPnP.sequence.status.nextStep := #JOB_1_STEP_13;
   END_IF;
END_REGION

REGION Network 21: Step[113] : Main P&P 1 Rotary Cylinder InHomePos
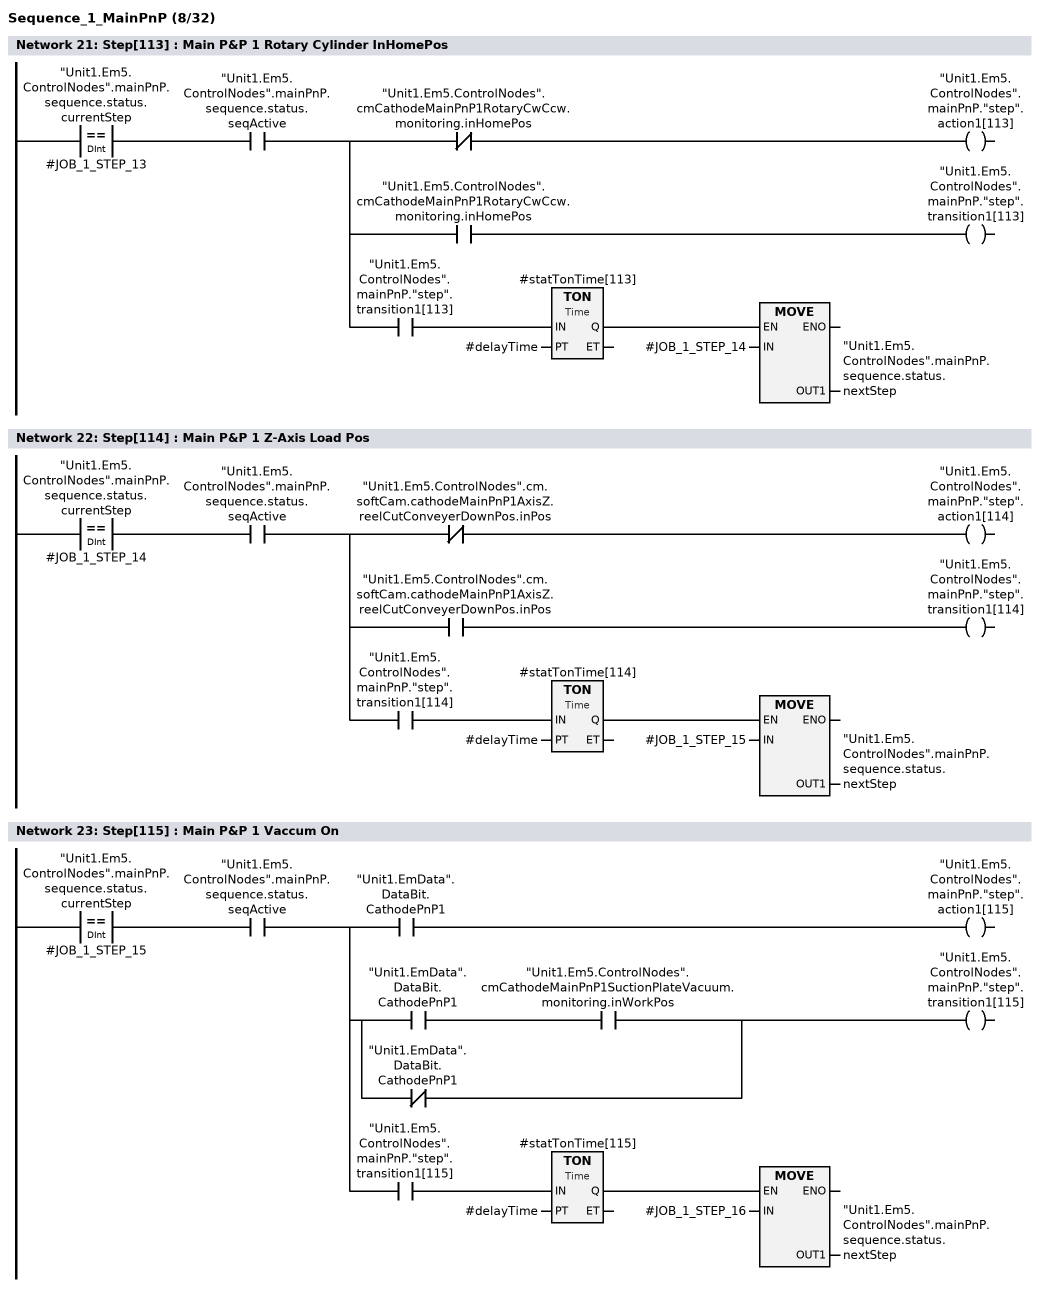
   RUNG wire#powerrail
      { S7_Templates := "SrcType := DInt" } EQ_Contact(in1 := "Unit1.Em5.ControlNodes".mainPnP.sequence.status.currentStep, in2 := #JOB_1_STEP_13)
      Contact( "Unit1.Em5.ControlNodes".mainPnP.sequence.status.seqActive )
      wire#w1
      I_Contact( "Unit1.Em5.ControlNodes".cmCathodeMainPnP1RotaryCwCcw.monitoring.inHomePos )
      Coil( "Unit1.Em5.ControlNodes".mainPnP."step".action1[113] )
   END_RUNG
   RUNG wire#w1
      Contact( "Unit1.Em5.ControlNodes".cmCathodeMainPnP1RotaryCwCcw.monitoring.inHomePos )
      Coil( "Unit1.Em5.ControlNodes".mainPnP."step".transition1[113] )
   END_RUNG
   RUNG wire#w1
      Contact( "Unit1.Em5.ControlNodes".mainPnP."step".transition1[113] )
      { S7_Templates := "time_type := Time" } #statTonTime[113].TON(pt := #delayTime, et =>)
      Move(in := #JOB_1_STEP_14, out1 => "Unit1.Em5.ControlNodes".mainPnP.sequence.status.nextStep)
   END_RUNG
   // the same network as SCL:
   #_w1 := ("Unit1.Em5.ControlNodes".mainPnP.sequence.status.currentStep = #JOB_1_STEP_13) AND "Unit1.Em5.ControlNodes".mainPnP.sequence.status.seqActive;
   "Unit1.Em5.ControlNodes".mainPnP."step".action1[113] := #_w1 AND NOT "Unit1.Em5.ControlNodes".cmCathodeMainPnP1RotaryCwCcw.monitoring.inHomePos;
   "Unit1.Em5.ControlNodes".mainPnP."step".transition1[113] := #_w1 AND "Unit1.Em5.ControlNodes".cmCathodeMainPnP1RotaryCwCcw.monitoring.inHomePos;
   #statTonTime[113].TON(IN := #_w1 AND "Unit1.Em5.ControlNodes".mainPnP."step".transition1[113],
                         PT := #delayTime);
   IF #statTonTime[113].Q THEN
       "Unit1.Em5.ControlNodes".mainPnP.sequence.status.nextStep := #JOB_1_STEP_14;
   END_IF;
END_REGION

REGION Network 22: Step[114] : Main P&P 1 Z-Axis Load Pos
   RUNG wire#powerrail
      { S7_Templates := "SrcType := DInt" } EQ_Contact(in1 := "Unit1.Em5.ControlNodes".mainPnP.sequence.status.currentStep, in2 := #JOB_1_STEP_14)
      Contact( "Unit1.Em5.ControlNodes".mainPnP.sequence.status.seqActive )
      wire#w1
      I_Contact( "Unit1.Em5.ControlNodes".cm.softCam.cathodeMainPnP1AxisZ.reelCutConveyerDownPos.inPos )
      Coil( "Unit1.Em5.ControlNodes".mainPnP."step".action1[114] )
   END_RUNG
   RUNG wire#w1
      Contact( "Unit1.Em5.ControlNodes".cm.softCam.cathodeMainPnP1AxisZ.reelCutConveyerDownPos.inPos )
      Coil( "Unit1.Em5.ControlNodes".mainPnP."step".transition1[114] )
   END_RUNG
   RUNG wire#w1
      Contact( "Unit1.Em5.ControlNodes".mainPnP."step".transition1[114] )
      { S7_Templates := "time_type := Time" } #statTonTime[114].TON(pt := #delayTime, et =>)
      Move(in := #JOB_1_STEP_15, out1 => "Unit1.Em5.ControlNodes".mainPnP.sequence.status.nextStep)
   END_RUNG
   // the same network as SCL:
   #_w1 := ("Unit1.Em5.ControlNodes".mainPnP.sequence.status.currentStep = #JOB_1_STEP_14) AND "Unit1.Em5.ControlNodes".mainPnP.sequence.status.seqActive;
   "Unit1.Em5.ControlNodes".mainPnP."step".action1[114] := #_w1 AND NOT "Unit1.Em5.ControlNodes".cm.softCam.cathodeMainPnP1AxisZ.reelCutConveyerDownPos.inPos;
   "Unit1.Em5.ControlNodes".mainPnP."step".transition1[114] := #_w1 AND "Unit1.Em5.ControlNodes".cm.softCam.cathodeMainPnP1AxisZ.reelCutConveyerDownPos.inPos;
   #statTonTime[114].TON(IN := #_w1 AND "Unit1.Em5.ControlNodes".mainPnP."step".transition1[114],
                         PT := #delayTime);
   IF #statTonTime[114].Q THEN
       "Unit1.Em5.ControlNodes".mainPnP.sequence.status.nextStep := #JOB_1_STEP_15;
   END_IF;
END_REGION

REGION Network 23: Step[115] : Main P&P 1 Vaccum On
   RUNG wire#powerrail
      { S7_Templates := "SrcType := DInt" } EQ_Contact(in1 := "Unit1.Em5.ControlNodes".mainPnP.sequence.status.currentStep, in2 := #JOB_1_STEP_15)
      Contact( "Unit1.Em5.ControlNodes".mainPnP.sequence.status.seqActive )
      wire#w1
      Contact( "Unit1.EmData".DataBit.CathodePnP1 )
      Coil( "Unit1.Em5.ControlNodes".mainPnP."step".action1[115] )
   END_RUNG
   RUNG wire#w1
      Contact( "Unit1.EmData".DataBit.CathodePnP1 )
      Contact( "Unit1.Em5.ControlNodes".cmCathodeMainPnP1SuctionPlateVacuum.monitoring.inWorkPos )
      wire#w2
      Coil( "Unit1.Em5.ControlNodes".mainPnP."step".transition1[115] )
   END_RUNG
   RUNG wire#w1
      I_Contact( "Unit1.EmData".DataBit.CathodePnP1 )
   END_RUNG wire#w2
   RUNG wire#w1
      Contact( "Unit1.Em5.ControlNodes".mainPnP."step".transition1[115] )
      { S7_Templates := "time_type := Time" } #statTonTime[115].TON(pt := #delayTime, et =>)
      Move(in := #JOB_1_STEP_16, out1 => "Unit1.Em5.ControlNodes".mainPnP.sequence.status.nextStep)
   END_RUNG
   // the same network as SCL:
   #_w1 := ("Unit1.Em5.ControlNodes".mainPnP.sequence.status.currentStep = #JOB_1_STEP_15) AND "Unit1.Em5.ControlNodes".mainPnP.sequence.status.seqActive;
   "Unit1.Em5.ControlNodes".mainPnP."step".action1[115] := #_w1 AND "Unit1.EmData".DataBit.CathodePnP1;
   "Unit1.Em5.ControlNodes".mainPnP."step".transition1[115] := #_w1 AND (("Unit1.EmData".DataBit.CathodePnP1 AND "Unit1.Em5.ControlNodes".cmCathodeMainPnP1SuctionPlateVacuum.monitoring.inWorkPos) OR NOT "Unit1.EmData".DataBit.CathodePnP1);
   #statTonTime[115].TON(IN := #_w1 AND "Unit1.Em5.ControlNodes".mainPnP."step".transition1[115],
                         PT := #delayTime);
   IF #statTonTime[115].Q THEN
       "Unit1.Em5.ControlNodes".mainPnP.sequence.status.nextStep := #JOB_1_STEP_16;
   END_IF;
END_REGION

REGION Network 24: Step[116] : Main P&P 1 Pick Up Blow On
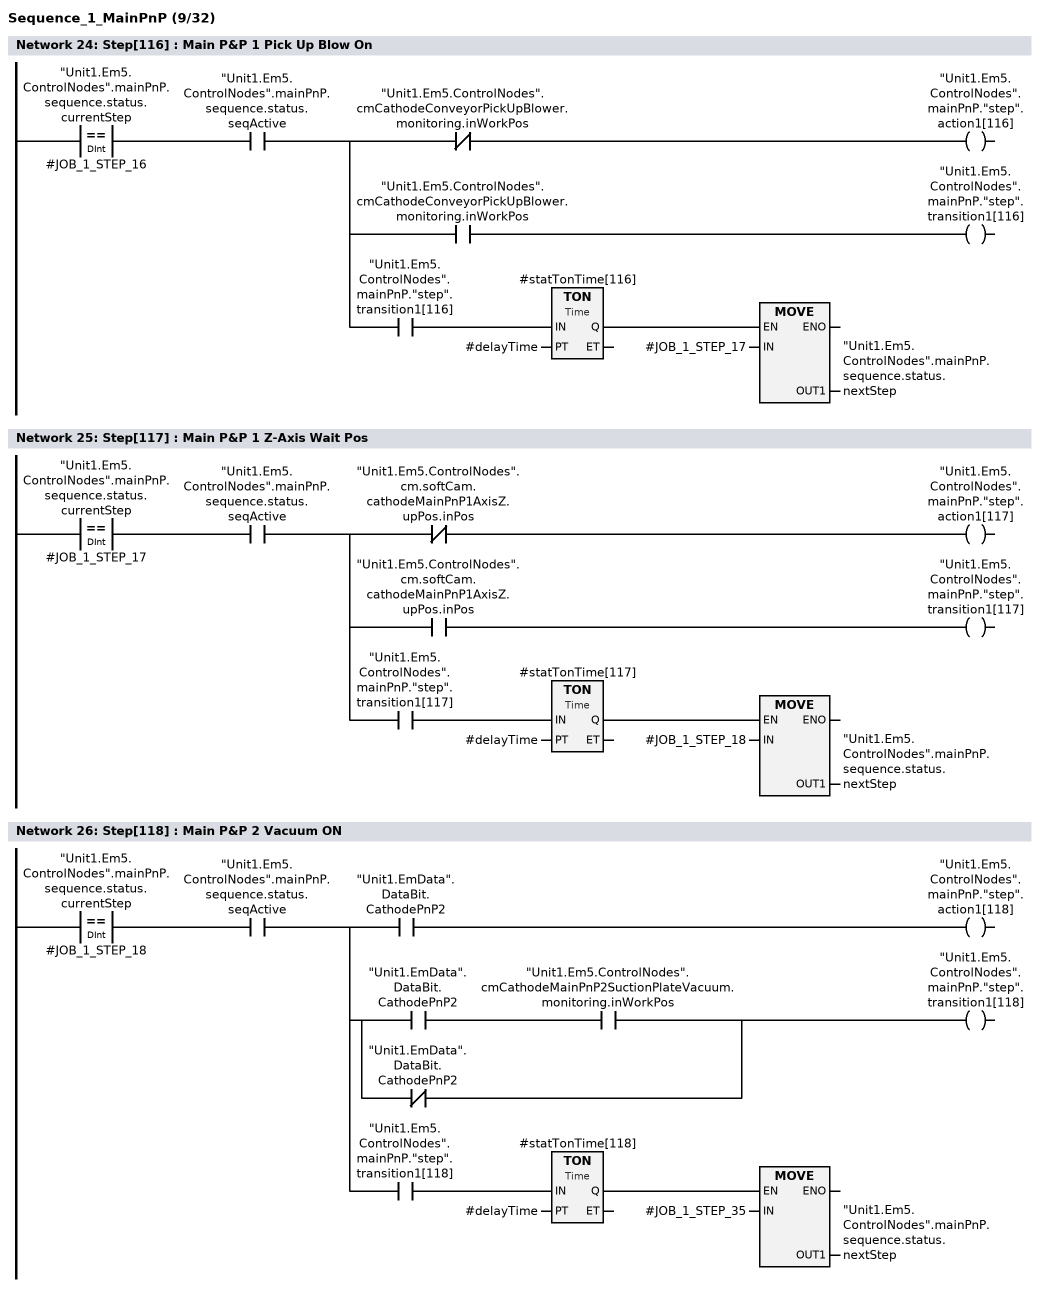
   RUNG wire#powerrail
      { S7_Templates := "SrcType := DInt" } EQ_Contact(in1 := "Unit1.Em5.ControlNodes".mainPnP.sequence.status.currentStep, in2 := #JOB_1_STEP_16)
      Contact( "Unit1.Em5.ControlNodes".mainPnP.sequence.status.seqActive )
      wire#w1
      I_Contact( "Unit1.Em5.ControlNodes".cmCathodeConveyorPickUpBlower.monitoring.inWorkPos )
      Coil( "Unit1.Em5.ControlNodes".mainPnP."step".action1[116] )
   END_RUNG
   RUNG wire#w1
      Contact( "Unit1.Em5.ControlNodes".cmCathodeConveyorPickUpBlower.monitoring.inWorkPos )
      Coil( "Unit1.Em5.ControlNodes".mainPnP."step".transition1[116] )
   END_RUNG
   RUNG wire#w1
      Contact( "Unit1.Em5.ControlNodes".mainPnP."step".transition1[116] )
      { S7_Templates := "time_type := Time" } #statTonTime[116].TON(pt := #delayTime, et =>)
      Move(in := #JOB_1_STEP_17, out1 => "Unit1.Em5.ControlNodes".mainPnP.sequence.status.nextStep)
   END_RUNG
   // the same network as SCL:
   #_w1 := ("Unit1.Em5.ControlNodes".mainPnP.sequence.status.currentStep = #JOB_1_STEP_16) AND "Unit1.Em5.ControlNodes".mainPnP.sequence.status.seqActive;
   "Unit1.Em5.ControlNodes".mainPnP."step".action1[116] := #_w1 AND NOT "Unit1.Em5.ControlNodes".cmCathodeConveyorPickUpBlower.monitoring.inWorkPos;
   "Unit1.Em5.ControlNodes".mainPnP."step".transition1[116] := #_w1 AND "Unit1.Em5.ControlNodes".cmCathodeConveyorPickUpBlower.monitoring.inWorkPos;
   #statTonTime[116].TON(IN := #_w1 AND "Unit1.Em5.ControlNodes".mainPnP."step".transition1[116],
                         PT := #delayTime);
   IF #statTonTime[116].Q THEN
       "Unit1.Em5.ControlNodes".mainPnP.sequence.status.nextStep := #JOB_1_STEP_17;
   END_IF;
END_REGION

REGION Network 25: Step[117] : Main P&P 1 Z-Axis Wait Pos
   RUNG wire#powerrail
      { S7_Templates := "SrcType := DInt" } EQ_Contact(in1 := "Unit1.Em5.ControlNodes".mainPnP.sequence.status.currentStep, in2 := #JOB_1_STEP_17)
      Contact( "Unit1.Em5.ControlNodes".mainPnP.sequence.status.seqActive )
      wire#w1
      I_Contact( "Unit1.Em5.ControlNodes".cm.softCam.cathodeMainPnP1AxisZ.upPos.inPos )
      Coil( "Unit1.Em5.ControlNodes".mainPnP."step".action1[117] )
   END_RUNG
   RUNG wire#w1
      Contact( "Unit1.Em5.ControlNodes".cm.softCam.cathodeMainPnP1AxisZ.upPos.inPos )
      Coil( "Unit1.Em5.ControlNodes".mainPnP."step".transition1[117] )
   END_RUNG
   RUNG wire#w1
      Contact( "Unit1.Em5.ControlNodes".mainPnP."step".transition1[117] )
      { S7_Templates := "time_type := Time" } #statTonTime[117].TON(pt := #delayTime, et =>)
      Move(in := #JOB_1_STEP_18, out1 => "Unit1.Em5.ControlNodes".mainPnP.sequence.status.nextStep)
   END_RUNG
   // the same network as SCL:
   #_w1 := ("Unit1.Em5.ControlNodes".mainPnP.sequence.status.currentStep = #JOB_1_STEP_17) AND "Unit1.Em5.ControlNodes".mainPnP.sequence.status.seqActive;
   "Unit1.Em5.ControlNodes".mainPnP."step".action1[117] := #_w1 AND NOT "Unit1.Em5.ControlNodes".cm.softCam.cathodeMainPnP1AxisZ.upPos.inPos;
   "Unit1.Em5.ControlNodes".mainPnP."step".transition1[117] := #_w1 AND "Unit1.Em5.ControlNodes".cm.softCam.cathodeMainPnP1AxisZ.upPos.inPos;
   #statTonTime[117].TON(IN := #_w1 AND "Unit1.Em5.ControlNodes".mainPnP."step".transition1[117],
                         PT := #delayTime);
   IF #statTonTime[117].Q THEN
       "Unit1.Em5.ControlNodes".mainPnP.sequence.status.nextStep := #JOB_1_STEP_18;
   END_IF;
END_REGION

REGION Network 26: Step[118] : Main P&P 2 Vacuum ON
   RUNG wire#powerrail
      { S7_Templates := "SrcType := DInt" } EQ_Contact(in1 := "Unit1.Em5.ControlNodes".mainPnP.sequence.status.currentStep, in2 := #JOB_1_STEP_18)
      Contact( "Unit1.Em5.ControlNodes".mainPnP.sequence.status.seqActive )
      wire#w1
      Contact( "Unit1.EmData".DataBit.CathodePnP2 )
      Coil( "Unit1.Em5.ControlNodes".mainPnP."step".action1[118] )
   END_RUNG
   RUNG wire#w1
      Contact( "Unit1.EmData".DataBit.CathodePnP2 )
      Contact( "Unit1.Em5.ControlNodes".cmCathodeMainPnP2SuctionPlateVacuum.monitoring.inWorkPos )
      wire#w2
      Coil( "Unit1.Em5.ControlNodes".mainPnP."step".transition1[118] )
   END_RUNG
   RUNG wire#w1
      I_Contact( "Unit1.EmData".DataBit.CathodePnP2 )
   END_RUNG wire#w2
   RUNG wire#w1
      Contact( "Unit1.Em5.ControlNodes".mainPnP."step".transition1[118] )
      { S7_Templates := "time_type := Time" } #statTonTime[118].TON(pt := #delayTime, et =>)
      Move(in := #JOB_1_STEP_35, out1 => "Unit1.Em5.ControlNodes".mainPnP.sequence.status.nextStep)
   END_RUNG
   // the same network as SCL:
   #_w1 := ("Unit1.Em5.ControlNodes".mainPnP.sequence.status.currentStep = #JOB_1_STEP_18) AND "Unit1.Em5.ControlNodes".mainPnP.sequence.status.seqActive;
   "Unit1.Em5.ControlNodes".mainPnP."step".action1[118] := #_w1 AND "Unit1.EmData".DataBit.CathodePnP2;
   "Unit1.Em5.ControlNodes".mainPnP."step".transition1[118] := #_w1 AND (("Unit1.EmData".DataBit.CathodePnP2 AND "Unit1.Em5.ControlNodes".cmCathodeMainPnP2SuctionPlateVacuum.monitoring.inWorkPos) OR NOT "Unit1.EmData".DataBit.CathodePnP2);
   #statTonTime[118].TON(IN := #_w1 AND "Unit1.Em5.ControlNodes".mainPnP."step".transition1[118],
                         PT := #delayTime);
   IF #statTonTime[118].Q THEN
       "Unit1.Em5.ControlNodes".mainPnP.sequence.status.nextStep := #JOB_1_STEP_35;
   END_IF;
END_REGION

REGION Network 28: Step[120] : Main P&P 1,2 X-Axis Unload Pos
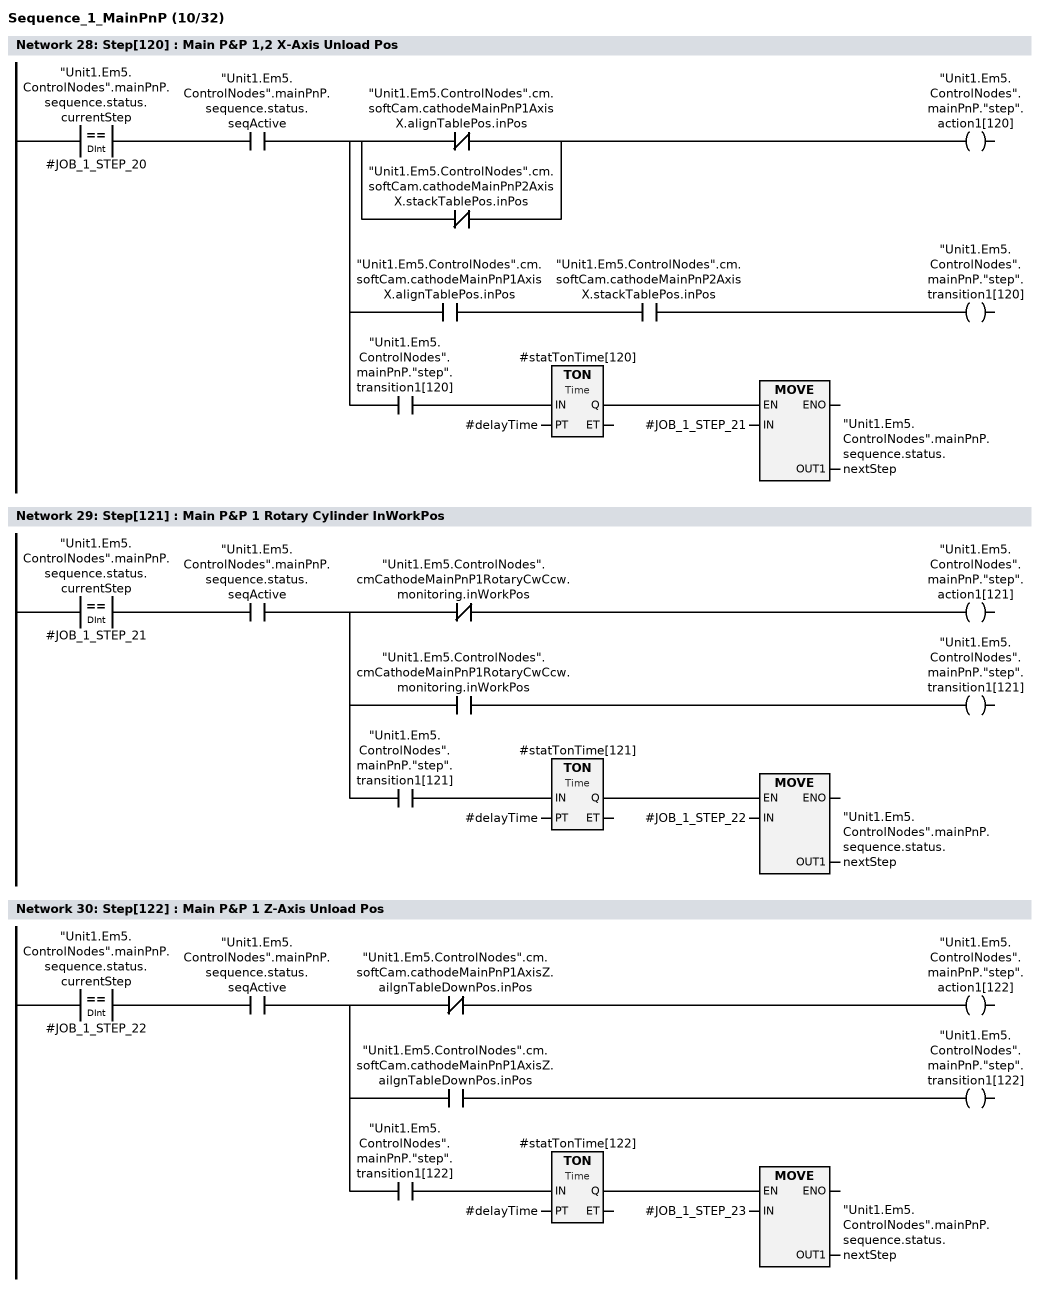
   RUNG wire#powerrail
      { S7_Templates := "SrcType := DInt" } EQ_Contact(in1 := "Unit1.Em5.ControlNodes".mainPnP.sequence.status.currentStep, in2 := #JOB_1_STEP_20)
      Contact( "Unit1.Em5.ControlNodes".mainPnP.sequence.status.seqActive )
      wire#w1
      I_Contact( "Unit1.Em5.ControlNodes".cm.softCam.cathodeMainPnP1AxisX.alignTablePos.inPos )
      wire#w2
      Coil( "Unit1.Em5.ControlNodes".mainPnP."step".action1[120] )
   END_RUNG
   RUNG wire#w1
      I_Contact( "Unit1.Em5.ControlNodes".cm.softCam.cathodeMainPnP2AxisX.stackTablePos.inPos )
   END_RUNG wire#w2
   RUNG wire#w1
      Contact( "Unit1.Em5.ControlNodes".cm.softCam.cathodeMainPnP1AxisX.alignTablePos.inPos )
      Contact( "Unit1.Em5.ControlNodes".cm.softCam.cathodeMainPnP2AxisX.stackTablePos.inPos )
      Coil( "Unit1.Em5.ControlNodes".mainPnP."step".transition1[120] )
   END_RUNG
   RUNG wire#w1
      Contact( "Unit1.Em5.ControlNodes".mainPnP."step".transition1[120] )
      { S7_Templates := "time_type := Time" } #statTonTime[120].TON(pt := #delayTime, et =>)
      Move(in := #JOB_1_STEP_21, out1 => "Unit1.Em5.ControlNodes".mainPnP.sequence.status.nextStep)
   END_RUNG
   // the same network as SCL:
   #_w1 := ("Unit1.Em5.ControlNodes".mainPnP.sequence.status.currentStep = #JOB_1_STEP_20) AND "Unit1.Em5.ControlNodes".mainPnP.sequence.status.seqActive;
   "Unit1.Em5.ControlNodes".mainPnP."step".action1[120] := #_w1 AND (NOT "Unit1.Em5.ControlNodes".cm.softCam.cathodeMainPnP1AxisX.alignTablePos.inPos OR NOT "Unit1.Em5.ControlNodes".cm.softCam.cathodeMainPnP2AxisX.stackTablePos.inPos);
   "Unit1.Em5.ControlNodes".mainPnP."step".transition1[120] := #_w1 AND "Unit1.Em5.ControlNodes".cm.softCam.cathodeMainPnP1AxisX.alignTablePos.inPos AND "Unit1.Em5.ControlNodes".cm.softCam.cathodeMainPnP2AxisX.stackTablePos.inPos;
   #statTonTime[120].TON(IN := #_w1 AND "Unit1.Em5.ControlNodes".mainPnP."step".transition1[120],
                         PT := #delayTime);
   IF #statTonTime[120].Q THEN
       "Unit1.Em5.ControlNodes".mainPnP.sequence.status.nextStep := #JOB_1_STEP_21;
   END_IF;
END_REGION

REGION Network 29: Step[121] : Main P&P 1 Rotary Cylinder InWorkPos
   RUNG wire#powerrail
      { S7_Templates := "SrcType := DInt" } EQ_Contact(in1 := "Unit1.Em5.ControlNodes".mainPnP.sequence.status.currentStep, in2 := #JOB_1_STEP_21)
      Contact( "Unit1.Em5.ControlNodes".mainPnP.sequence.status.seqActive )
      wire#w1
      I_Contact( "Unit1.Em5.ControlNodes".cmCathodeMainPnP1RotaryCwCcw.monitoring.inWorkPos )
      Coil( "Unit1.Em5.ControlNodes".mainPnP."step".action1[121] )
   END_RUNG
   RUNG wire#w1
      Contact( "Unit1.Em5.ControlNodes".cmCathodeMainPnP1RotaryCwCcw.monitoring.inWorkPos )
      Coil( "Unit1.Em5.ControlNodes".mainPnP."step".transition1[121] )
   END_RUNG
   RUNG wire#w1
      Contact( "Unit1.Em5.ControlNodes".mainPnP."step".transition1[121] )
      { S7_Templates := "time_type := Time" } #statTonTime[121].TON(pt := #delayTime, et =>)
      Move(in := #JOB_1_STEP_22, out1 => "Unit1.Em5.ControlNodes".mainPnP.sequence.status.nextStep)
   END_RUNG
   // the same network as SCL:
   #_w1 := ("Unit1.Em5.ControlNodes".mainPnP.sequence.status.currentStep = #JOB_1_STEP_21) AND "Unit1.Em5.ControlNodes".mainPnP.sequence.status.seqActive;
   "Unit1.Em5.ControlNodes".mainPnP."step".action1[121] := #_w1 AND NOT "Unit1.Em5.ControlNodes".cmCathodeMainPnP1RotaryCwCcw.monitoring.inWorkPos;
   "Unit1.Em5.ControlNodes".mainPnP."step".transition1[121] := #_w1 AND "Unit1.Em5.ControlNodes".cmCathodeMainPnP1RotaryCwCcw.monitoring.inWorkPos;
   #statTonTime[121].TON(IN := #_w1 AND "Unit1.Em5.ControlNodes".mainPnP."step".transition1[121],
                         PT := #delayTime);
   IF #statTonTime[121].Q THEN
       "Unit1.Em5.ControlNodes".mainPnP.sequence.status.nextStep := #JOB_1_STEP_22;
   END_IF;
END_REGION

REGION Network 30: Step[122] : Main P&P 1 Z-Axis Unload Pos
   RUNG wire#powerrail
      { S7_Templates := "SrcType := DInt" } EQ_Contact(in1 := "Unit1.Em5.ControlNodes".mainPnP.sequence.status.currentStep, in2 := #JOB_1_STEP_22)
      Contact( "Unit1.Em5.ControlNodes".mainPnP.sequence.status.seqActive )
      wire#w1
      I_Contact( "Unit1.Em5.ControlNodes".cm.softCam.cathodeMainPnP1AxisZ.ailgnTableDownPos.inPos )
      Coil( "Unit1.Em5.ControlNodes".mainPnP."step".action1[122] )
   END_RUNG
   RUNG wire#w1
      Contact( "Unit1.Em5.ControlNodes".cm.softCam.cathodeMainPnP1AxisZ.ailgnTableDownPos.inPos )
      Coil( "Unit1.Em5.ControlNodes".mainPnP."step".transition1[122] )
   END_RUNG
   RUNG wire#w1
      Contact( "Unit1.Em5.ControlNodes".mainPnP."step".transition1[122] )
      { S7_Templates := "time_type := Time" } #statTonTime[122].TON(pt := #delayTime, et =>)
      Move(in := #JOB_1_STEP_23, out1 => "Unit1.Em5.ControlNodes".mainPnP.sequence.status.nextStep)
   END_RUNG
   // the same network as SCL:
   #_w1 := ("Unit1.Em5.ControlNodes".mainPnP.sequence.status.currentStep = #JOB_1_STEP_22) AND "Unit1.Em5.ControlNodes".mainPnP.sequence.status.seqActive;
   "Unit1.Em5.ControlNodes".mainPnP."step".action1[122] := #_w1 AND NOT "Unit1.Em5.ControlNodes".cm.softCam.cathodeMainPnP1AxisZ.ailgnTableDownPos.inPos;
   "Unit1.Em5.ControlNodes".mainPnP."step".transition1[122] := #_w1 AND "Unit1.Em5.ControlNodes".cm.softCam.cathodeMainPnP1AxisZ.ailgnTableDownPos.inPos;
   #statTonTime[122].TON(IN := #_w1 AND "Unit1.Em5.ControlNodes".mainPnP."step".transition1[122],
                         PT := #delayTime);
   IF #statTonTime[122].Q THEN
       "Unit1.Em5.ControlNodes".mainPnP.sequence.status.nextStep := #JOB_1_STEP_23;
   END_IF;
END_REGION

REGION Network 31: Step[123] : Main P&P → Align Table [Unloading Ready]
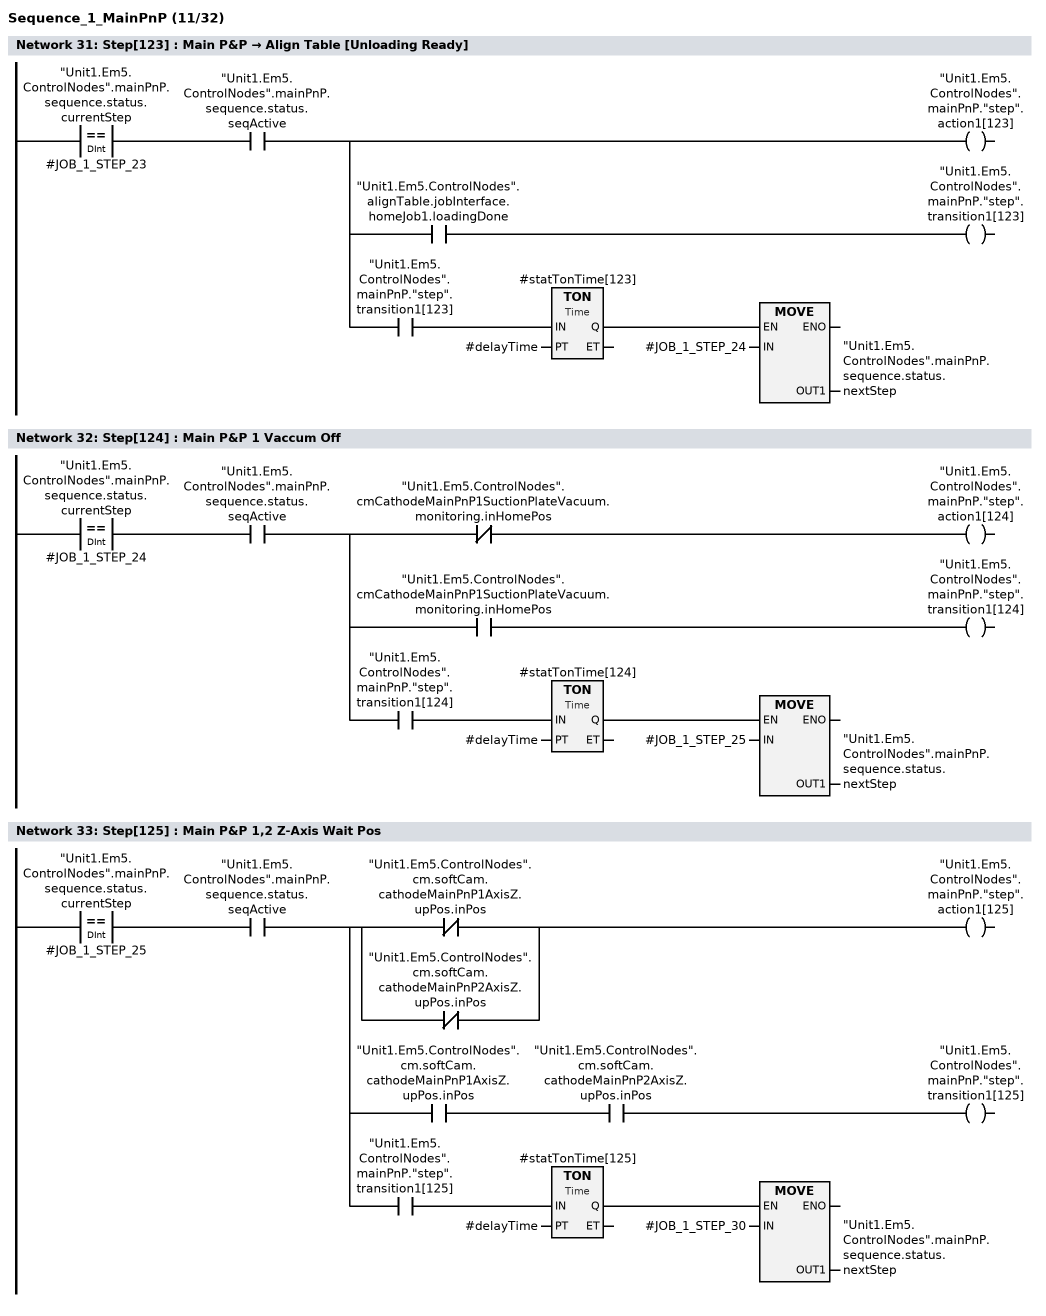
   RUNG wire#powerrail
      { S7_Templates := "SrcType := DInt" } EQ_Contact(in1 := "Unit1.Em5.ControlNodes".mainPnP.sequence.status.currentStep, in2 := #JOB_1_STEP_23)
      Contact( "Unit1.Em5.ControlNodes".mainPnP.sequence.status.seqActive )
      wire#w1
      Coil( "Unit1.Em5.ControlNodes".mainPnP."step".action1[123] )
   END_RUNG
   RUNG wire#w1
      Contact( "Unit1.Em5.ControlNodes".alignTable.jobInterface.homeJob1.loadingDone )
      Coil( "Unit1.Em5.ControlNodes".mainPnP."step".transition1[123] )
   END_RUNG
   RUNG wire#w1
      Contact( "Unit1.Em5.ControlNodes".mainPnP."step".transition1[123] )
      { S7_Templates := "time_type := Time" } #statTonTime[123].TON(pt := #delayTime, et =>)
      Move(in := #JOB_1_STEP_24, out1 => "Unit1.Em5.ControlNodes".mainPnP.sequence.status.nextStep)
   END_RUNG
   // the same network as SCL:
   "Unit1.Em5.ControlNodes".mainPnP."step".action1[123] := ("Unit1.Em5.ControlNodes".mainPnP.sequence.status.currentStep = #JOB_1_STEP_23) AND "Unit1.Em5.ControlNodes".mainPnP.sequence.status.seqActive;
   "Unit1.Em5.ControlNodes".mainPnP."step".transition1[123] := ("Unit1.Em5.ControlNodes".mainPnP.sequence.status.currentStep = #JOB_1_STEP_23) AND "Unit1.Em5.ControlNodes".mainPnP.sequence.status.seqActive AND "Unit1.Em5.ControlNodes".alignTable.jobInterface.homeJob1.loadingDone;
   #statTonTime[123].TON(IN := ("Unit1.Em5.ControlNodes".mainPnP.sequence.status.currentStep = #JOB_1_STEP_23) AND "Unit1.Em5.ControlNodes".mainPnP.sequence.status.seqActive AND "Unit1.Em5.ControlNodes".mainPnP."step".transition1[123],
                         PT := #delayTime);
   IF #statTonTime[123].Q THEN
       "Unit1.Em5.ControlNodes".mainPnP.sequence.status.nextStep := #JOB_1_STEP_24;
   END_IF;
END_REGION

REGION Network 32: Step[124] : Main P&P 1 Vaccum Off
   RUNG wire#powerrail
      { S7_Templates := "SrcType := DInt" } EQ_Contact(in1 := "Unit1.Em5.ControlNodes".mainPnP.sequence.status.currentStep, in2 := #JOB_1_STEP_24)
      Contact( "Unit1.Em5.ControlNodes".mainPnP.sequence.status.seqActive )
      wire#w1
      I_Contact( "Unit1.Em5.ControlNodes".cmCathodeMainPnP1SuctionPlateVacuum.monitoring.inHomePos )
      Coil( "Unit1.Em5.ControlNodes".mainPnP."step".action1[124] )
   END_RUNG
   RUNG wire#w1
      Contact( "Unit1.Em5.ControlNodes".cmCathodeMainPnP1SuctionPlateVacuum.monitoring.inHomePos )
      Coil( "Unit1.Em5.ControlNodes".mainPnP."step".transition1[124] )
   END_RUNG
   RUNG wire#w1
      Contact( "Unit1.Em5.ControlNodes".mainPnP."step".transition1[124] )
      { S7_Templates := "time_type := Time" } #statTonTime[124].TON(pt := #delayTime, et =>)
      Move(in := #JOB_1_STEP_25, out1 => "Unit1.Em5.ControlNodes".mainPnP.sequence.status.nextStep)
   END_RUNG
   // the same network as SCL:
   #_w1 := ("Unit1.Em5.ControlNodes".mainPnP.sequence.status.currentStep = #JOB_1_STEP_24) AND "Unit1.Em5.ControlNodes".mainPnP.sequence.status.seqActive;
   "Unit1.Em5.ControlNodes".mainPnP."step".action1[124] := #_w1 AND NOT "Unit1.Em5.ControlNodes".cmCathodeMainPnP1SuctionPlateVacuum.monitoring.inHomePos;
   "Unit1.Em5.ControlNodes".mainPnP."step".transition1[124] := #_w1 AND "Unit1.Em5.ControlNodes".cmCathodeMainPnP1SuctionPlateVacuum.monitoring.inHomePos;
   #statTonTime[124].TON(IN := #_w1 AND "Unit1.Em5.ControlNodes".mainPnP."step".transition1[124],
                         PT := #delayTime);
   IF #statTonTime[124].Q THEN
       "Unit1.Em5.ControlNodes".mainPnP.sequence.status.nextStep := #JOB_1_STEP_25;
   END_IF;
END_REGION

REGION Network 33: Step[125] : Main P&P 1,2 Z-Axis Wait Pos
   RUNG wire#powerrail
      { S7_Templates := "SrcType := DInt" } EQ_Contact(in1 := "Unit1.Em5.ControlNodes".mainPnP.sequence.status.currentStep, in2 := #JOB_1_STEP_25)
      Contact( "Unit1.Em5.ControlNodes".mainPnP.sequence.status.seqActive )
      wire#w1
      I_Contact( "Unit1.Em5.ControlNodes".cm.softCam.cathodeMainPnP1AxisZ.upPos.inPos )
      wire#w2
      Coil( "Unit1.Em5.ControlNodes".mainPnP."step".action1[125] )
   END_RUNG
   RUNG wire#w1
      I_Contact( "Unit1.Em5.ControlNodes".cm.softCam.cathodeMainPnP2AxisZ.upPos.inPos )
   END_RUNG wire#w2
   RUNG wire#w1
      Contact( "Unit1.Em5.ControlNodes".cm.softCam.cathodeMainPnP1AxisZ.upPos.inPos )
      Contact( "Unit1.Em5.ControlNodes".cm.softCam.cathodeMainPnP2AxisZ.upPos.inPos )
      Coil( "Unit1.Em5.ControlNodes".mainPnP."step".transition1[125] )
   END_RUNG
   RUNG wire#w1
      Contact( "Unit1.Em5.ControlNodes".mainPnP."step".transition1[125] )
      { S7_Templates := "time_type := Time" } #statTonTime[125].TON(pt := #delayTime, et =>)
      Move(in := #JOB_1_STEP_30, out1 => "Unit1.Em5.ControlNodes".mainPnP.sequence.status.nextStep)
   END_RUNG
   // the same network as SCL:
   #_w1 := ("Unit1.Em5.ControlNodes".mainPnP.sequence.status.currentStep = #JOB_1_STEP_25) AND "Unit1.Em5.ControlNodes".mainPnP.sequence.status.seqActive;
   "Unit1.Em5.ControlNodes".mainPnP."step".action1[125] := #_w1 AND (NOT "Unit1.Em5.ControlNodes".cm.softCam.cathodeMainPnP1AxisZ.upPos.inPos OR NOT "Unit1.Em5.ControlNodes".cm.softCam.cathodeMainPnP2AxisZ.upPos.inPos);
   "Unit1.Em5.ControlNodes".mainPnP."step".transition1[125] := #_w1 AND "Unit1.Em5.ControlNodes".cm.softCam.cathodeMainPnP1AxisZ.upPos.inPos AND "Unit1.Em5.ControlNodes".cm.softCam.cathodeMainPnP2AxisZ.upPos.inPos;
   #statTonTime[125].TON(IN := #_w1 AND "Unit1.Em5.ControlNodes".mainPnP."step".transition1[125],
                         PT := #delayTime);
   IF #statTonTime[125].Q THEN
       "Unit1.Em5.ControlNodes".mainPnP.sequence.status.nextStep := #JOB_1_STEP_30;
   END_IF;
END_REGION

REGION Network 35: Step[130] : Main P&P 1,2 X-Axis Load Pos
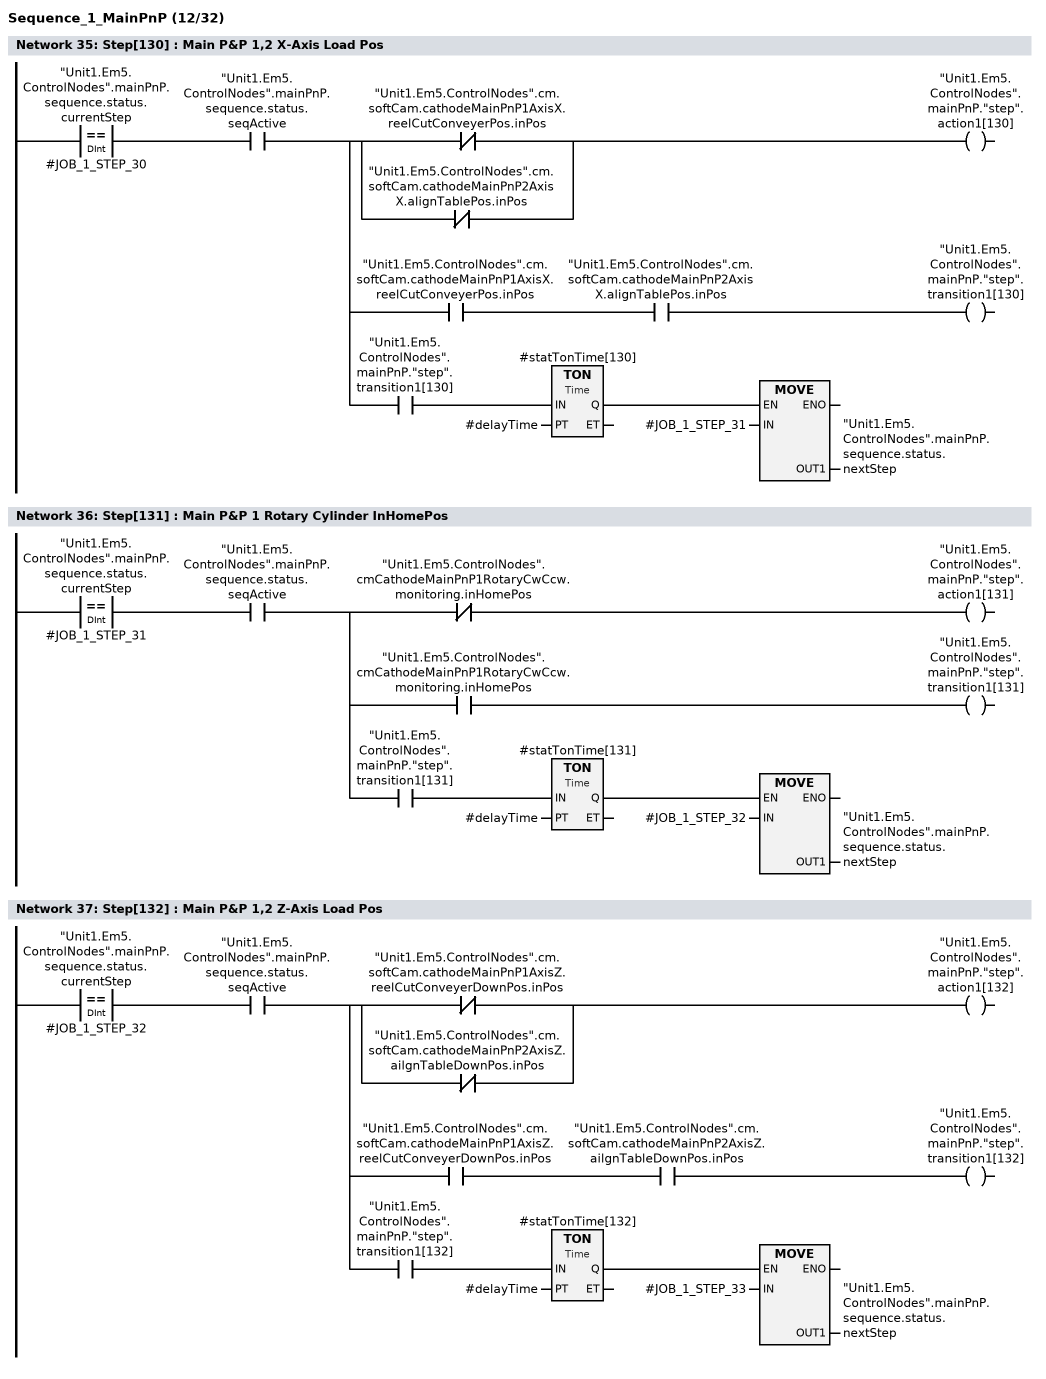
   RUNG wire#powerrail
      { S7_Templates := "SrcType := DInt" } EQ_Contact(in1 := "Unit1.Em5.ControlNodes".mainPnP.sequence.status.currentStep, in2 := #JOB_1_STEP_30)
      Contact( "Unit1.Em5.ControlNodes".mainPnP.sequence.status.seqActive )
      wire#w1
      I_Contact( "Unit1.Em5.ControlNodes".cm.softCam.cathodeMainPnP1AxisX.reelCutConveyerPos.inPos )
      wire#w2
      Coil( "Unit1.Em5.ControlNodes".mainPnP."step".action1[130] )
   END_RUNG
   RUNG wire#w1
      I_Contact( "Unit1.Em5.ControlNodes".cm.softCam.cathodeMainPnP2AxisX.alignTablePos.inPos )
   END_RUNG wire#w2
   RUNG wire#w1
      Contact( "Unit1.Em5.ControlNodes".cm.softCam.cathodeMainPnP1AxisX.reelCutConveyerPos.inPos )
      Contact( "Unit1.Em5.ControlNodes".cm.softCam.cathodeMainPnP2AxisX.alignTablePos.inPos )
      Coil( "Unit1.Em5.ControlNodes".mainPnP."step".transition1[130] )
   END_RUNG
   RUNG wire#w1
      Contact( "Unit1.Em5.ControlNodes".mainPnP."step".transition1[130] )
      { S7_Templates := "time_type := Time" } #statTonTime[130].TON(pt := #delayTime, et =>)
      Move(in := #JOB_1_STEP_31, out1 => "Unit1.Em5.ControlNodes".mainPnP.sequence.status.nextStep)
   END_RUNG
   // the same network as SCL:
   #_w1 := ("Unit1.Em5.ControlNodes".mainPnP.sequence.status.currentStep = #JOB_1_STEP_30) AND "Unit1.Em5.ControlNodes".mainPnP.sequence.status.seqActive;
   "Unit1.Em5.ControlNodes".mainPnP."step".action1[130] := #_w1 AND (NOT "Unit1.Em5.ControlNodes".cm.softCam.cathodeMainPnP1AxisX.reelCutConveyerPos.inPos OR NOT "Unit1.Em5.ControlNodes".cm.softCam.cathodeMainPnP2AxisX.alignTablePos.inPos);
   "Unit1.Em5.ControlNodes".mainPnP."step".transition1[130] := #_w1 AND "Unit1.Em5.ControlNodes".cm.softCam.cathodeMainPnP1AxisX.reelCutConveyerPos.inPos AND "Unit1.Em5.ControlNodes".cm.softCam.cathodeMainPnP2AxisX.alignTablePos.inPos;
   #statTonTime[130].TON(IN := #_w1 AND "Unit1.Em5.ControlNodes".mainPnP."step".transition1[130],
                         PT := #delayTime);
   IF #statTonTime[130].Q THEN
       "Unit1.Em5.ControlNodes".mainPnP.sequence.status.nextStep := #JOB_1_STEP_31;
   END_IF;
END_REGION

REGION Network 36: Step[131] : Main P&P 1 Rotary Cylinder InHomePos
   RUNG wire#powerrail
      { S7_Templates := "SrcType := DInt" } EQ_Contact(in1 := "Unit1.Em5.ControlNodes".mainPnP.sequence.status.currentStep, in2 := #JOB_1_STEP_31)
      Contact( "Unit1.Em5.ControlNodes".mainPnP.sequence.status.seqActive )
      wire#w1
      I_Contact( "Unit1.Em5.ControlNodes".cmCathodeMainPnP1RotaryCwCcw.monitoring.inHomePos )
      Coil( "Unit1.Em5.ControlNodes".mainPnP."step".action1[131] )
   END_RUNG
   RUNG wire#w1
      Contact( "Unit1.Em5.ControlNodes".cmCathodeMainPnP1RotaryCwCcw.monitoring.inHomePos )
      Coil( "Unit1.Em5.ControlNodes".mainPnP."step".transition1[131] )
   END_RUNG
   RUNG wire#w1
      Contact( "Unit1.Em5.ControlNodes".mainPnP."step".transition1[131] )
      { S7_Templates := "time_type := Time" } #statTonTime[131].TON(pt := #delayTime, et =>)
      Move(in := #JOB_1_STEP_32, out1 => "Unit1.Em5.ControlNodes".mainPnP.sequence.status.nextStep)
   END_RUNG
   // the same network as SCL:
   #_w1 := ("Unit1.Em5.ControlNodes".mainPnP.sequence.status.currentStep = #JOB_1_STEP_31) AND "Unit1.Em5.ControlNodes".mainPnP.sequence.status.seqActive;
   "Unit1.Em5.ControlNodes".mainPnP."step".action1[131] := #_w1 AND NOT "Unit1.Em5.ControlNodes".cmCathodeMainPnP1RotaryCwCcw.monitoring.inHomePos;
   "Unit1.Em5.ControlNodes".mainPnP."step".transition1[131] := #_w1 AND "Unit1.Em5.ControlNodes".cmCathodeMainPnP1RotaryCwCcw.monitoring.inHomePos;
   #statTonTime[131].TON(IN := #_w1 AND "Unit1.Em5.ControlNodes".mainPnP."step".transition1[131],
                         PT := #delayTime);
   IF #statTonTime[131].Q THEN
       "Unit1.Em5.ControlNodes".mainPnP.sequence.status.nextStep := #JOB_1_STEP_32;
   END_IF;
END_REGION

REGION Network 37: Step[132] : Main P&P 1,2 Z-Axis Load Pos
   RUNG wire#powerrail
      { S7_Templates := "SrcType := DInt" } EQ_Contact(in1 := "Unit1.Em5.ControlNodes".mainPnP.sequence.status.currentStep, in2 := #JOB_1_STEP_32)
      Contact( "Unit1.Em5.ControlNodes".mainPnP.sequence.status.seqActive )
      wire#w1
      I_Contact( "Unit1.Em5.ControlNodes".cm.softCam.cathodeMainPnP1AxisZ.reelCutConveyerDownPos.inPos )
      wire#w2
      Coil( "Unit1.Em5.ControlNodes".mainPnP."step".action1[132] )
   END_RUNG
   RUNG wire#w1
      I_Contact( "Unit1.Em5.ControlNodes".cm.softCam.cathodeMainPnP2AxisZ.ailgnTableDownPos.inPos )
   END_RUNG wire#w2
   RUNG wire#w1
      Contact( "Unit1.Em5.ControlNodes".cm.softCam.cathodeMainPnP1AxisZ.reelCutConveyerDownPos.inPos )
      Contact( "Unit1.Em5.ControlNodes".cm.softCam.cathodeMainPnP2AxisZ.ailgnTableDownPos.inPos )
      Coil( "Unit1.Em5.ControlNodes".mainPnP."step".transition1[132] )
   END_RUNG
   RUNG wire#w1
      Contact( "Unit1.Em5.ControlNodes".mainPnP."step".transition1[132] )
      { S7_Templates := "time_type := Time" } #statTonTime[132].TON(pt := #delayTime, et =>)
      Move(in := #JOB_1_STEP_33, out1 => "Unit1.Em5.ControlNodes".mainPnP.sequence.status.nextStep)
   END_RUNG
   // the same network as SCL:
   #_w1 := ("Unit1.Em5.ControlNodes".mainPnP.sequence.status.currentStep = #JOB_1_STEP_32) AND "Unit1.Em5.ControlNodes".mainPnP.sequence.status.seqActive;
   "Unit1.Em5.ControlNodes".mainPnP."step".action1[132] := #_w1 AND (NOT "Unit1.Em5.ControlNodes".cm.softCam.cathodeMainPnP1AxisZ.reelCutConveyerDownPos.inPos OR NOT "Unit1.Em5.ControlNodes".cm.softCam.cathodeMainPnP2AxisZ.ailgnTableDownPos.inPos);
   "Unit1.Em5.ControlNodes".mainPnP."step".transition1[132] := #_w1 AND "Unit1.Em5.ControlNodes".cm.softCam.cathodeMainPnP1AxisZ.reelCutConveyerDownPos.inPos AND "Unit1.Em5.ControlNodes".cm.softCam.cathodeMainPnP2AxisZ.ailgnTableDownPos.inPos;
   #statTonTime[132].TON(IN := #_w1 AND "Unit1.Em5.ControlNodes".mainPnP."step".transition1[132],
                         PT := #delayTime);
   IF #statTonTime[132].Q THEN
       "Unit1.Em5.ControlNodes".mainPnP.sequence.status.nextStep := #JOB_1_STEP_33;
   END_IF;
END_REGION

REGION Network 38: Step[133] : Main P&P 1,2 Vaccum On
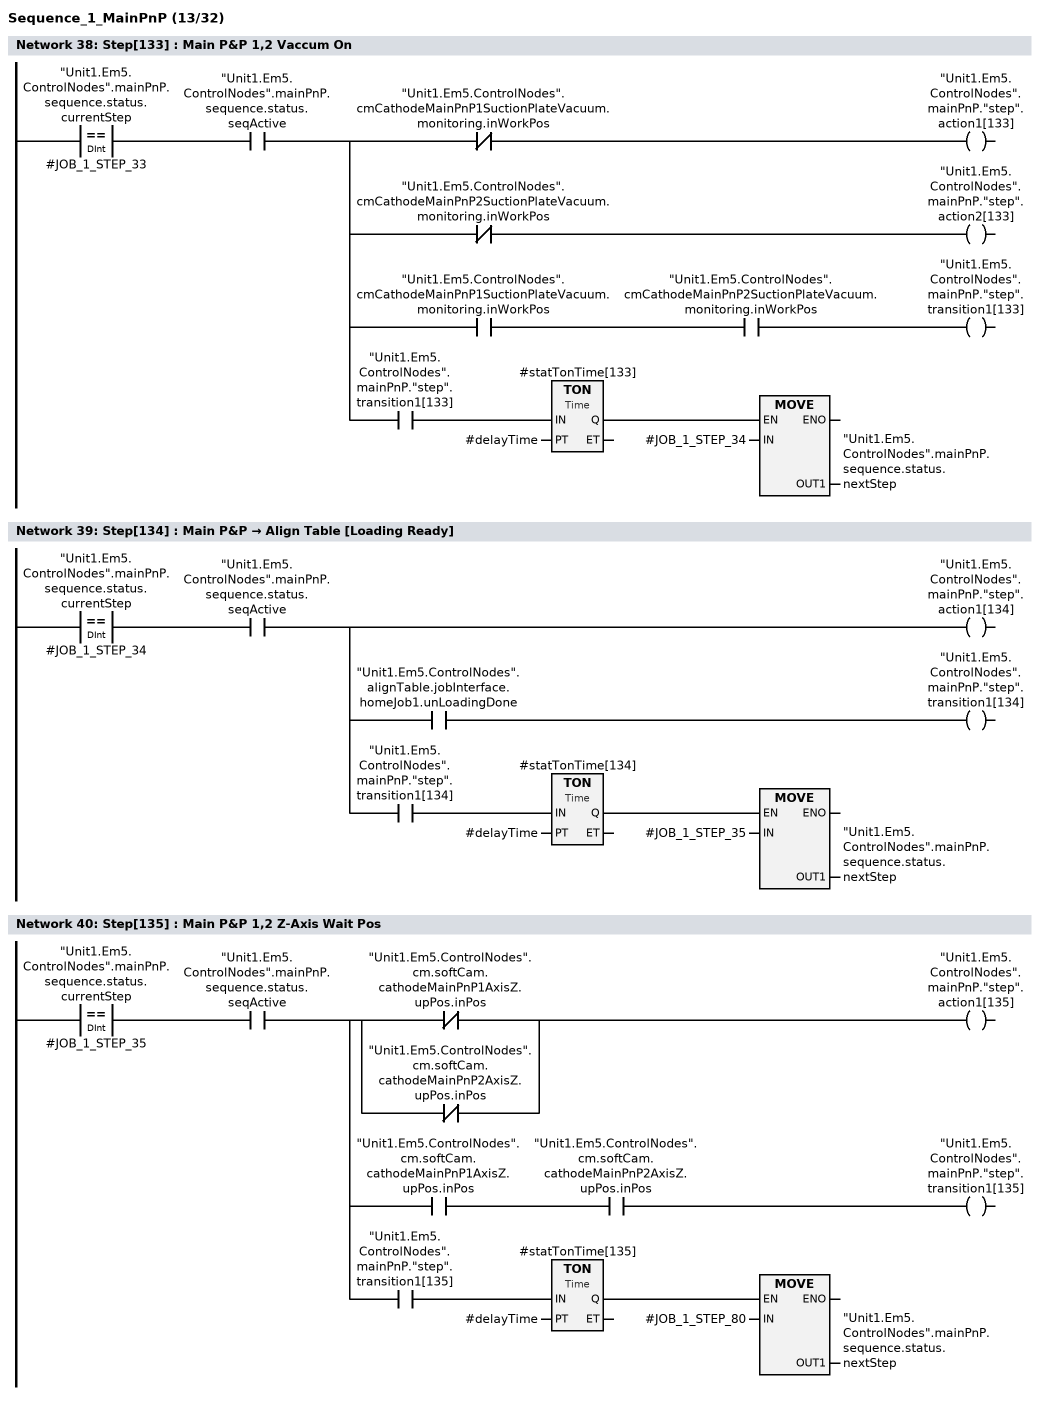
   RUNG wire#powerrail
      { S7_Templates := "SrcType := DInt" } EQ_Contact(in1 := "Unit1.Em5.ControlNodes".mainPnP.sequence.status.currentStep, in2 := #JOB_1_STEP_33)
      Contact( "Unit1.Em5.ControlNodes".mainPnP.sequence.status.seqActive )
      wire#w1
      I_Contact( "Unit1.Em5.ControlNodes".cmCathodeMainPnP1SuctionPlateVacuum.monitoring.inWorkPos )
      Coil( "Unit1.Em5.ControlNodes".mainPnP."step".action1[133] )
   END_RUNG
   RUNG wire#w1
      I_Contact( "Unit1.Em5.ControlNodes".cmCathodeMainPnP2SuctionPlateVacuum.monitoring.inWorkPos )
      Coil( "Unit1.Em5.ControlNodes".mainPnP."step".action2[133] )
   END_RUNG
   RUNG wire#w1
      Contact( "Unit1.Em5.ControlNodes".cmCathodeMainPnP1SuctionPlateVacuum.monitoring.inWorkPos )
      Contact( "Unit1.Em5.ControlNodes".cmCathodeMainPnP2SuctionPlateVacuum.monitoring.inWorkPos )
      Coil( "Unit1.Em5.ControlNodes".mainPnP."step".transition1[133] )
   END_RUNG
   RUNG wire#w1
      Contact( "Unit1.Em5.ControlNodes".mainPnP."step".transition1[133] )
      { S7_Templates := "time_type := Time" } #statTonTime[133].TON(pt := #delayTime, et =>)
      Move(in := #JOB_1_STEP_34, out1 => "Unit1.Em5.ControlNodes".mainPnP.sequence.status.nextStep)
   END_RUNG
   // the same network as SCL:
   #_w1 := ("Unit1.Em5.ControlNodes".mainPnP.sequence.status.currentStep = #JOB_1_STEP_33) AND "Unit1.Em5.ControlNodes".mainPnP.sequence.status.seqActive;
   "Unit1.Em5.ControlNodes".mainPnP."step".action1[133] := #_w1 AND NOT "Unit1.Em5.ControlNodes".cmCathodeMainPnP1SuctionPlateVacuum.monitoring.inWorkPos;
   "Unit1.Em5.ControlNodes".mainPnP."step".action2[133] := #_w1 AND NOT "Unit1.Em5.ControlNodes".cmCathodeMainPnP2SuctionPlateVacuum.monitoring.inWorkPos;
   "Unit1.Em5.ControlNodes".mainPnP."step".transition1[133] := #_w1 AND "Unit1.Em5.ControlNodes".cmCathodeMainPnP1SuctionPlateVacuum.monitoring.inWorkPos AND "Unit1.Em5.ControlNodes".cmCathodeMainPnP2SuctionPlateVacuum.monitoring.inWorkPos;
   #statTonTime[133].TON(IN := #_w1 AND "Unit1.Em5.ControlNodes".mainPnP."step".transition1[133],
                         PT := #delayTime);
   IF #statTonTime[133].Q THEN
       "Unit1.Em5.ControlNodes".mainPnP.sequence.status.nextStep := #JOB_1_STEP_34;
   END_IF;
END_REGION

REGION Network 39: Step[134] : Main P&P → Align Table [Loading Ready]
   RUNG wire#powerrail
      { S7_Templates := "SrcType := DInt" } EQ_Contact(in1 := "Unit1.Em5.ControlNodes".mainPnP.sequence.status.currentStep, in2 := #JOB_1_STEP_34)
      Contact( "Unit1.Em5.ControlNodes".mainPnP.sequence.status.seqActive )
      wire#w1
      Coil( "Unit1.Em5.ControlNodes".mainPnP."step".action1[134] )
   END_RUNG
   RUNG wire#w1
      Contact( "Unit1.Em5.ControlNodes".alignTable.jobInterface.homeJob1.unLoadingDone )
      Coil( "Unit1.Em5.ControlNodes".mainPnP."step".transition1[134] )
   END_RUNG
   RUNG wire#w1
      Contact( "Unit1.Em5.ControlNodes".mainPnP."step".transition1[134] )
      { S7_Templates := "time_type := Time" } #statTonTime[134].TON(pt := #delayTime, et =>)
      Move(in := #JOB_1_STEP_35, out1 => "Unit1.Em5.ControlNodes".mainPnP.sequence.status.nextStep)
   END_RUNG
   // the same network as SCL:
   "Unit1.Em5.ControlNodes".mainPnP."step".action1[134] := ("Unit1.Em5.ControlNodes".mainPnP.sequence.status.currentStep = #JOB_1_STEP_34) AND "Unit1.Em5.ControlNodes".mainPnP.sequence.status.seqActive;
   "Unit1.Em5.ControlNodes".mainPnP."step".transition1[134] := ("Unit1.Em5.ControlNodes".mainPnP.sequence.status.currentStep = #JOB_1_STEP_34) AND "Unit1.Em5.ControlNodes".mainPnP.sequence.status.seqActive AND "Unit1.Em5.ControlNodes".alignTable.jobInterface.homeJob1.unLoadingDone;
   #statTonTime[134].TON(IN := ("Unit1.Em5.ControlNodes".mainPnP.sequence.status.currentStep = #JOB_1_STEP_34) AND "Unit1.Em5.ControlNodes".mainPnP.sequence.status.seqActive AND "Unit1.Em5.ControlNodes".mainPnP."step".transition1[134],
                         PT := #delayTime);
   IF #statTonTime[134].Q THEN
       "Unit1.Em5.ControlNodes".mainPnP.sequence.status.nextStep := #JOB_1_STEP_35;
   END_IF;
END_REGION

REGION Network 40: Step[135] : Main P&P 1,2 Z-Axis Wait Pos
   RUNG wire#powerrail
      { S7_Templates := "SrcType := DInt" } EQ_Contact(in1 := "Unit1.Em5.ControlNodes".mainPnP.sequence.status.currentStep, in2 := #JOB_1_STEP_35)
      Contact( "Unit1.Em5.ControlNodes".mainPnP.sequence.status.seqActive )
      wire#w1
      I_Contact( "Unit1.Em5.ControlNodes".cm.softCam.cathodeMainPnP1AxisZ.upPos.inPos )
      wire#w2
      Coil( "Unit1.Em5.ControlNodes".mainPnP."step".action1[135] )
   END_RUNG
   RUNG wire#w1
      I_Contact( "Unit1.Em5.ControlNodes".cm.softCam.cathodeMainPnP2AxisZ.upPos.inPos )
   END_RUNG wire#w2
   RUNG wire#w1
      Contact( "Unit1.Em5.ControlNodes".cm.softCam.cathodeMainPnP1AxisZ.upPos.inPos )
      Contact( "Unit1.Em5.ControlNodes".cm.softCam.cathodeMainPnP2AxisZ.upPos.inPos )
      Coil( "Unit1.Em5.ControlNodes".mainPnP."step".transition1[135] )
   END_RUNG
   RUNG wire#w1
      Contact( "Unit1.Em5.ControlNodes".mainPnP."step".transition1[135] )
      { S7_Templates := "time_type := Time" } #statTonTime[135].TON(pt := #delayTime, et =>)
      Move(in := #JOB_1_STEP_80, out1 => "Unit1.Em5.ControlNodes".mainPnP.sequence.status.nextStep)
   END_RUNG
   // the same network as SCL:
   #_w1 := ("Unit1.Em5.ControlNodes".mainPnP.sequence.status.currentStep = #JOB_1_STEP_35) AND "Unit1.Em5.ControlNodes".mainPnP.sequence.status.seqActive;
   "Unit1.Em5.ControlNodes".mainPnP."step".action1[135] := #_w1 AND (NOT "Unit1.Em5.ControlNodes".cm.softCam.cathodeMainPnP1AxisZ.upPos.inPos OR NOT "Unit1.Em5.ControlNodes".cm.softCam.cathodeMainPnP2AxisZ.upPos.inPos);
   "Unit1.Em5.ControlNodes".mainPnP."step".transition1[135] := #_w1 AND "Unit1.Em5.ControlNodes".cm.softCam.cathodeMainPnP1AxisZ.upPos.inPos AND "Unit1.Em5.ControlNodes".cm.softCam.cathodeMainPnP2AxisZ.upPos.inPos;
   #statTonTime[135].TON(IN := #_w1 AND "Unit1.Em5.ControlNodes".mainPnP."step".transition1[135],
                         PT := #delayTime);
   IF #statTonTime[135].Q THEN
       "Unit1.Em5.ControlNodes".mainPnP.sequence.status.nextStep := #JOB_1_STEP_80;
   END_IF;
END_REGION

REGION Network 42: Step[140] : Main P&P 1,2 X-Axis Unload Pos
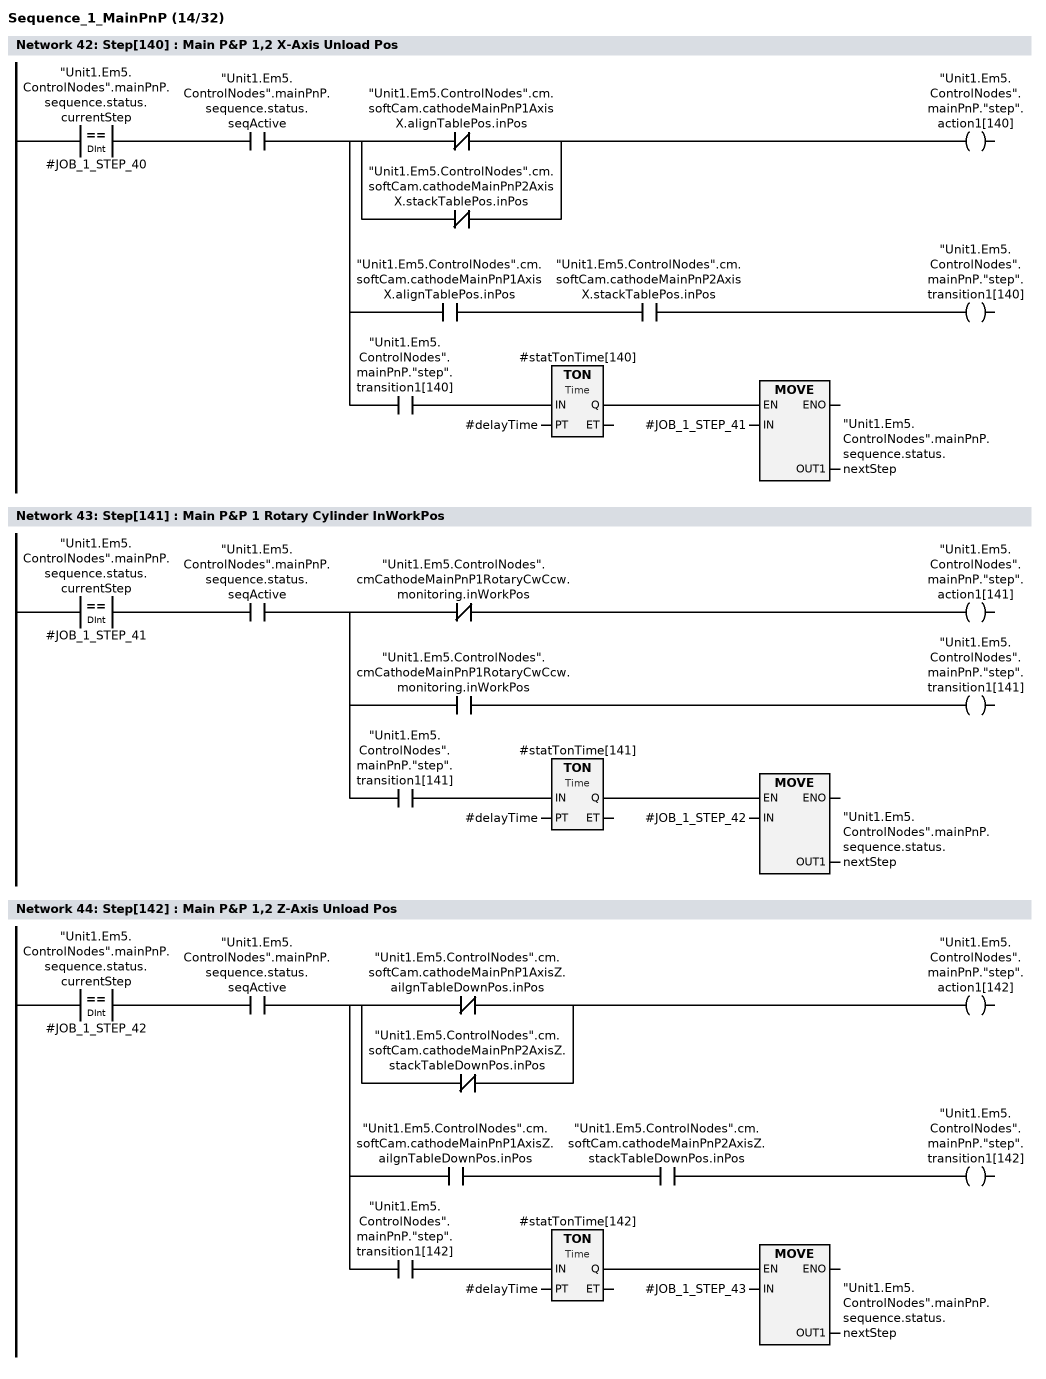
   RUNG wire#powerrail
      { S7_Templates := "SrcType := DInt" } EQ_Contact(in1 := "Unit1.Em5.ControlNodes".mainPnP.sequence.status.currentStep, in2 := #JOB_1_STEP_40)
      Contact( "Unit1.Em5.ControlNodes".mainPnP.sequence.status.seqActive )
      wire#w1
      I_Contact( "Unit1.Em5.ControlNodes".cm.softCam.cathodeMainPnP1AxisX.alignTablePos.inPos )
      wire#w2
      Coil( "Unit1.Em5.ControlNodes".mainPnP."step".action1[140] )
   END_RUNG
   RUNG wire#w1
      I_Contact( "Unit1.Em5.ControlNodes".cm.softCam.cathodeMainPnP2AxisX.stackTablePos.inPos )
   END_RUNG wire#w2
   RUNG wire#w1
      Contact( "Unit1.Em5.ControlNodes".cm.softCam.cathodeMainPnP1AxisX.alignTablePos.inPos )
      Contact( "Unit1.Em5.ControlNodes".cm.softCam.cathodeMainPnP2AxisX.stackTablePos.inPos )
      Coil( "Unit1.Em5.ControlNodes".mainPnP."step".transition1[140] )
   END_RUNG
   RUNG wire#w1
      Contact( "Unit1.Em5.ControlNodes".mainPnP."step".transition1[140] )
      { S7_Templates := "time_type := Time" } #statTonTime[140].TON(pt := #delayTime, et =>)
      Move(in := #JOB_1_STEP_41, out1 => "Unit1.Em5.ControlNodes".mainPnP.sequence.status.nextStep)
   END_RUNG
   // the same network as SCL:
   #_w1 := ("Unit1.Em5.ControlNodes".mainPnP.sequence.status.currentStep = #JOB_1_STEP_40) AND "Unit1.Em5.ControlNodes".mainPnP.sequence.status.seqActive;
   "Unit1.Em5.ControlNodes".mainPnP."step".action1[140] := #_w1 AND (NOT "Unit1.Em5.ControlNodes".cm.softCam.cathodeMainPnP1AxisX.alignTablePos.inPos OR NOT "Unit1.Em5.ControlNodes".cm.softCam.cathodeMainPnP2AxisX.stackTablePos.inPos);
   "Unit1.Em5.ControlNodes".mainPnP."step".transition1[140] := #_w1 AND "Unit1.Em5.ControlNodes".cm.softCam.cathodeMainPnP1AxisX.alignTablePos.inPos AND "Unit1.Em5.ControlNodes".cm.softCam.cathodeMainPnP2AxisX.stackTablePos.inPos;
   #statTonTime[140].TON(IN := #_w1 AND "Unit1.Em5.ControlNodes".mainPnP."step".transition1[140],
                         PT := #delayTime);
   IF #statTonTime[140].Q THEN
       "Unit1.Em5.ControlNodes".mainPnP.sequence.status.nextStep := #JOB_1_STEP_41;
   END_IF;
END_REGION

REGION Network 43: Step[141] : Main P&P 1 Rotary Cylinder InWorkPos
   RUNG wire#powerrail
      { S7_Templates := "SrcType := DInt" } EQ_Contact(in1 := "Unit1.Em5.ControlNodes".mainPnP.sequence.status.currentStep, in2 := #JOB_1_STEP_41)
      Contact( "Unit1.Em5.ControlNodes".mainPnP.sequence.status.seqActive )
      wire#w1
      I_Contact( "Unit1.Em5.ControlNodes".cmCathodeMainPnP1RotaryCwCcw.monitoring.inWorkPos )
      Coil( "Unit1.Em5.ControlNodes".mainPnP."step".action1[141] )
   END_RUNG
   RUNG wire#w1
      Contact( "Unit1.Em5.ControlNodes".cmCathodeMainPnP1RotaryCwCcw.monitoring.inWorkPos )
      Coil( "Unit1.Em5.ControlNodes".mainPnP."step".transition1[141] )
   END_RUNG
   RUNG wire#w1
      Contact( "Unit1.Em5.ControlNodes".mainPnP."step".transition1[141] )
      { S7_Templates := "time_type := Time" } #statTonTime[141].TON(pt := #delayTime, et =>)
      Move(in := #JOB_1_STEP_42, out1 => "Unit1.Em5.ControlNodes".mainPnP.sequence.status.nextStep)
   END_RUNG
   // the same network as SCL:
   #_w1 := ("Unit1.Em5.ControlNodes".mainPnP.sequence.status.currentStep = #JOB_1_STEP_41) AND "Unit1.Em5.ControlNodes".mainPnP.sequence.status.seqActive;
   "Unit1.Em5.ControlNodes".mainPnP."step".action1[141] := #_w1 AND NOT "Unit1.Em5.ControlNodes".cmCathodeMainPnP1RotaryCwCcw.monitoring.inWorkPos;
   "Unit1.Em5.ControlNodes".mainPnP."step".transition1[141] := #_w1 AND "Unit1.Em5.ControlNodes".cmCathodeMainPnP1RotaryCwCcw.monitoring.inWorkPos;
   #statTonTime[141].TON(IN := #_w1 AND "Unit1.Em5.ControlNodes".mainPnP."step".transition1[141],
                         PT := #delayTime);
   IF #statTonTime[141].Q THEN
       "Unit1.Em5.ControlNodes".mainPnP.sequence.status.nextStep := #JOB_1_STEP_42;
   END_IF;
END_REGION

REGION Network 44: Step[142] : Main P&P 1,2 Z-Axis Unload Pos
   RUNG wire#powerrail
      { S7_Templates := "SrcType := DInt" } EQ_Contact(in1 := "Unit1.Em5.ControlNodes".mainPnP.sequence.status.currentStep, in2 := #JOB_1_STEP_42)
      Contact( "Unit1.Em5.ControlNodes".mainPnP.sequence.status.seqActive )
      wire#w1
      I_Contact( "Unit1.Em5.ControlNodes".cm.softCam.cathodeMainPnP1AxisZ.ailgnTableDownPos.inPos )
      wire#w2
      Coil( "Unit1.Em5.ControlNodes".mainPnP."step".action1[142] )
   END_RUNG
   RUNG wire#w1
      I_Contact( "Unit1.Em5.ControlNodes".cm.softCam.cathodeMainPnP2AxisZ.stackTableDownPos.inPos )
   END_RUNG wire#w2
   RUNG wire#w1
      Contact( "Unit1.Em5.ControlNodes".cm.softCam.cathodeMainPnP1AxisZ.ailgnTableDownPos.inPos )
      Contact( "Unit1.Em5.ControlNodes".cm.softCam.cathodeMainPnP2AxisZ.stackTableDownPos.inPos )
      Coil( "Unit1.Em5.ControlNodes".mainPnP."step".transition1[142] )
   END_RUNG
   RUNG wire#w1
      Contact( "Unit1.Em5.ControlNodes".mainPnP."step".transition1[142] )
      { S7_Templates := "time_type := Time" } #statTonTime[142].TON(pt := #delayTime, et =>)
      Move(in := #JOB_1_STEP_43, out1 => "Unit1.Em5.ControlNodes".mainPnP.sequence.status.nextStep)
   END_RUNG
   // the same network as SCL:
   #_w1 := ("Unit1.Em5.ControlNodes".mainPnP.sequence.status.currentStep = #JOB_1_STEP_42) AND "Unit1.Em5.ControlNodes".mainPnP.sequence.status.seqActive;
   "Unit1.Em5.ControlNodes".mainPnP."step".action1[142] := #_w1 AND (NOT "Unit1.Em5.ControlNodes".cm.softCam.cathodeMainPnP1AxisZ.ailgnTableDownPos.inPos OR NOT "Unit1.Em5.ControlNodes".cm.softCam.cathodeMainPnP2AxisZ.stackTableDownPos.inPos);
   "Unit1.Em5.ControlNodes".mainPnP."step".transition1[142] := #_w1 AND "Unit1.Em5.ControlNodes".cm.softCam.cathodeMainPnP1AxisZ.ailgnTableDownPos.inPos AND "Unit1.Em5.ControlNodes".cm.softCam.cathodeMainPnP2AxisZ.stackTableDownPos.inPos;
   #statTonTime[142].TON(IN := #_w1 AND "Unit1.Em5.ControlNodes".mainPnP."step".transition1[142],
                         PT := #delayTime);
   IF #statTonTime[142].Q THEN
       "Unit1.Em5.ControlNodes".mainPnP.sequence.status.nextStep := #JOB_1_STEP_43;
   END_IF;
END_REGION

REGION Network 45: Step[143] : Main P&P → Align Table [Unloading Ready]
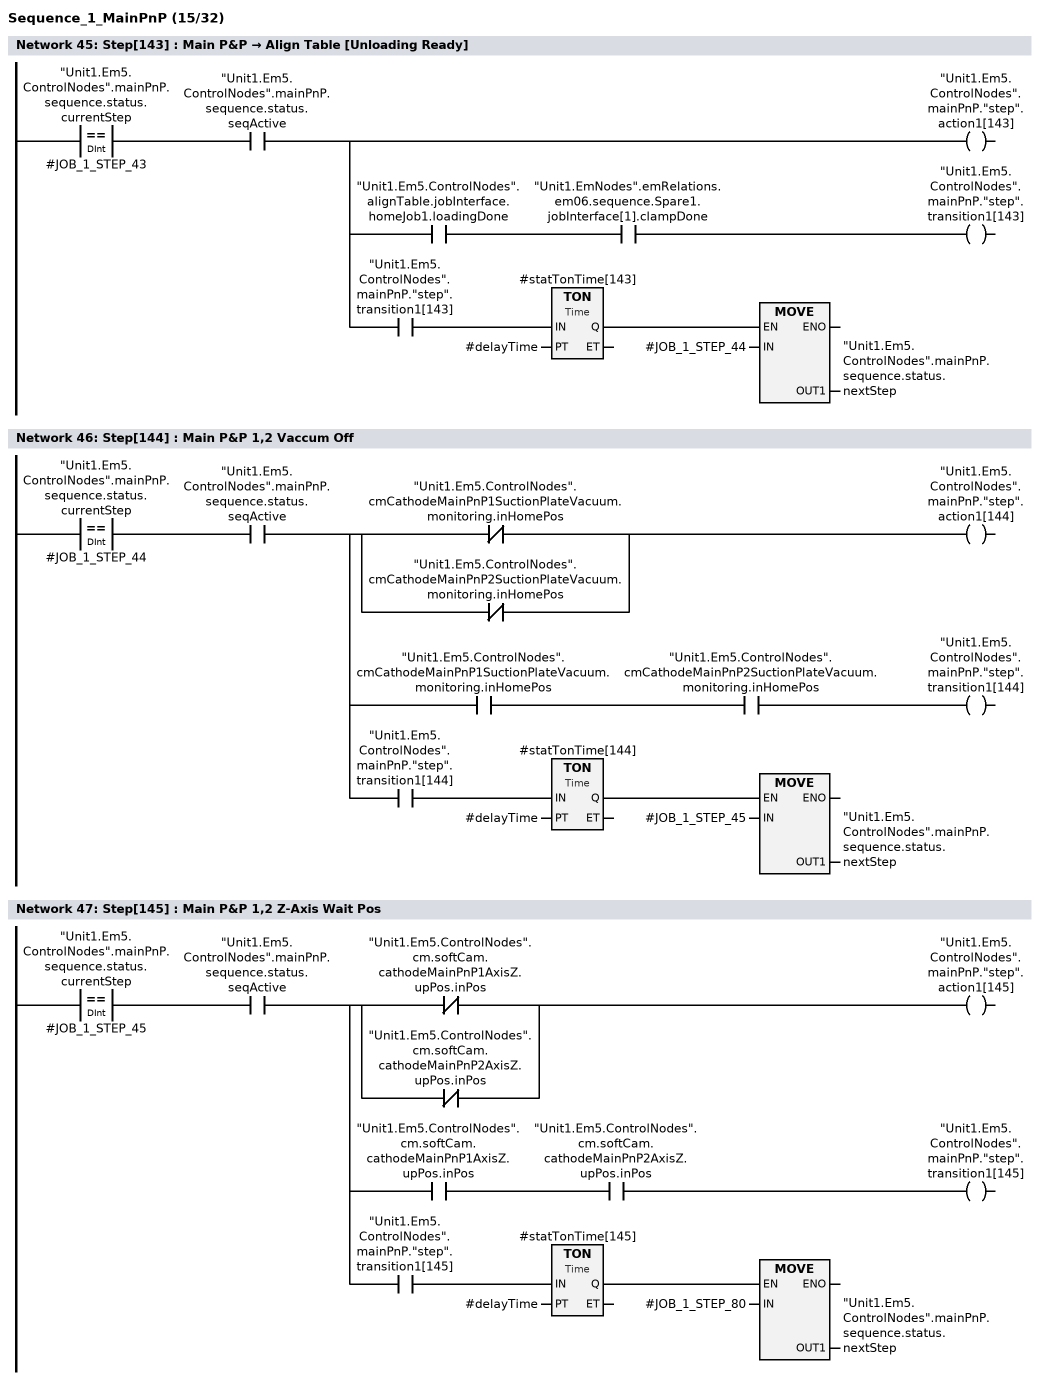
   RUNG wire#powerrail
      { S7_Templates := "SrcType := DInt" } EQ_Contact(in1 := "Unit1.Em5.ControlNodes".mainPnP.sequence.status.currentStep, in2 := #JOB_1_STEP_43)
      Contact( "Unit1.Em5.ControlNodes".mainPnP.sequence.status.seqActive )
      wire#w1
      Coil( "Unit1.Em5.ControlNodes".mainPnP."step".action1[143] )
   END_RUNG
   RUNG wire#w1
      Contact( "Unit1.Em5.ControlNodes".alignTable.jobInterface.homeJob1.loadingDone )
      Contact( "Unit1.EmNodes".emRelations.em06.sequence.Spare1.jobInterface[1].clampDone )
      Coil( "Unit1.Em5.ControlNodes".mainPnP."step".transition1[143] )
   END_RUNG
   RUNG wire#w1
      Contact( "Unit1.Em5.ControlNodes".mainPnP."step".transition1[143] )
      { S7_Templates := "time_type := Time" } #statTonTime[143].TON(pt := #delayTime, et =>)
      Move(in := #JOB_1_STEP_44, out1 => "Unit1.Em5.ControlNodes".mainPnP.sequence.status.nextStep)
   END_RUNG
   // the same network as SCL:
   "Unit1.Em5.ControlNodes".mainPnP."step".action1[143] := ("Unit1.Em5.ControlNodes".mainPnP.sequence.status.currentStep = #JOB_1_STEP_43) AND "Unit1.Em5.ControlNodes".mainPnP.sequence.status.seqActive;
   "Unit1.Em5.ControlNodes".mainPnP."step".transition1[143] := ("Unit1.Em5.ControlNodes".mainPnP.sequence.status.currentStep = #JOB_1_STEP_43) AND "Unit1.Em5.ControlNodes".mainPnP.sequence.status.seqActive AND "Unit1.Em5.ControlNodes".alignTable.jobInterface.homeJob1.loadingDone AND "Unit1.EmNodes".emRelations.em06.sequence.Spare1.jobInterface[1].clampDone;
   #statTonTime[143].TON(IN := ("Unit1.Em5.ControlNodes".mainPnP.sequence.status.currentStep = #JOB_1_STEP_43) AND "Unit1.Em5.ControlNodes".mainPnP.sequence.status.seqActive AND "Unit1.Em5.ControlNodes".mainPnP."step".transition1[143],
                         PT := #delayTime);
   IF #statTonTime[143].Q THEN
       "Unit1.Em5.ControlNodes".mainPnP.sequence.status.nextStep := #JOB_1_STEP_44;
   END_IF;
END_REGION

REGION Network 46: Step[144] : Main P&P 1,2 Vaccum Off
   RUNG wire#powerrail
      { S7_Templates := "SrcType := DInt" } EQ_Contact(in1 := "Unit1.Em5.ControlNodes".mainPnP.sequence.status.currentStep, in2 := #JOB_1_STEP_44)
      Contact( "Unit1.Em5.ControlNodes".mainPnP.sequence.status.seqActive )
      wire#w1
      I_Contact( "Unit1.Em5.ControlNodes".cmCathodeMainPnP1SuctionPlateVacuum.monitoring.inHomePos )
      wire#w2
      Coil( "Unit1.Em5.ControlNodes".mainPnP."step".action1[144] )
   END_RUNG
   RUNG wire#w1
      I_Contact( "Unit1.Em5.ControlNodes".cmCathodeMainPnP2SuctionPlateVacuum.monitoring.inHomePos )
   END_RUNG wire#w2
   RUNG wire#w1
      Contact( "Unit1.Em5.ControlNodes".cmCathodeMainPnP1SuctionPlateVacuum.monitoring.inHomePos )
      Contact( "Unit1.Em5.ControlNodes".cmCathodeMainPnP2SuctionPlateVacuum.monitoring.inHomePos )
      Coil( "Unit1.Em5.ControlNodes".mainPnP."step".transition1[144] )
   END_RUNG
   RUNG wire#w1
      Contact( "Unit1.Em5.ControlNodes".mainPnP."step".transition1[144] )
      { S7_Templates := "time_type := Time" } #statTonTime[144].TON(pt := #delayTime, et =>)
      Move(in := #JOB_1_STEP_45, out1 => "Unit1.Em5.ControlNodes".mainPnP.sequence.status.nextStep)
   END_RUNG
   // the same network as SCL:
   #_w1 := ("Unit1.Em5.ControlNodes".mainPnP.sequence.status.currentStep = #JOB_1_STEP_44) AND "Unit1.Em5.ControlNodes".mainPnP.sequence.status.seqActive;
   "Unit1.Em5.ControlNodes".mainPnP."step".action1[144] := #_w1 AND (NOT "Unit1.Em5.ControlNodes".cmCathodeMainPnP1SuctionPlateVacuum.monitoring.inHomePos OR NOT "Unit1.Em5.ControlNodes".cmCathodeMainPnP2SuctionPlateVacuum.monitoring.inHomePos);
   "Unit1.Em5.ControlNodes".mainPnP."step".transition1[144] := #_w1 AND "Unit1.Em5.ControlNodes".cmCathodeMainPnP1SuctionPlateVacuum.monitoring.inHomePos AND "Unit1.Em5.ControlNodes".cmCathodeMainPnP2SuctionPlateVacuum.monitoring.inHomePos;
   #statTonTime[144].TON(IN := #_w1 AND "Unit1.Em5.ControlNodes".mainPnP."step".transition1[144],
                         PT := #delayTime);
   IF #statTonTime[144].Q THEN
       "Unit1.Em5.ControlNodes".mainPnP.sequence.status.nextStep := #JOB_1_STEP_45;
   END_IF;
END_REGION

REGION Network 47: Step[145] : Main P&P 1,2 Z-Axis Wait Pos
   RUNG wire#powerrail
      { S7_Templates := "SrcType := DInt" } EQ_Contact(in1 := "Unit1.Em5.ControlNodes".mainPnP.sequence.status.currentStep, in2 := #JOB_1_STEP_45)
      Contact( "Unit1.Em5.ControlNodes".mainPnP.sequence.status.seqActive )
      wire#w1
      I_Contact( "Unit1.Em5.ControlNodes".cm.softCam.cathodeMainPnP1AxisZ.upPos.inPos )
      wire#w2
      Coil( "Unit1.Em5.ControlNodes".mainPnP."step".action1[145] )
   END_RUNG
   RUNG wire#w1
      I_Contact( "Unit1.Em5.ControlNodes".cm.softCam.cathodeMainPnP2AxisZ.upPos.inPos )
   END_RUNG wire#w2
   RUNG wire#w1
      Contact( "Unit1.Em5.ControlNodes".cm.softCam.cathodeMainPnP1AxisZ.upPos.inPos )
      Contact( "Unit1.Em5.ControlNodes".cm.softCam.cathodeMainPnP2AxisZ.upPos.inPos )
      Coil( "Unit1.Em5.ControlNodes".mainPnP."step".transition1[145] )
   END_RUNG
   RUNG wire#w1
      Contact( "Unit1.Em5.ControlNodes".mainPnP."step".transition1[145] )
      { S7_Templates := "time_type := Time" } #statTonTime[145].TON(pt := #delayTime, et =>)
      Move(in := #JOB_1_STEP_80, out1 => "Unit1.Em5.ControlNodes".mainPnP.sequence.status.nextStep)
   END_RUNG
   // the same network as SCL:
   #_w1 := ("Unit1.Em5.ControlNodes".mainPnP.sequence.status.currentStep = #JOB_1_STEP_45) AND "Unit1.Em5.ControlNodes".mainPnP.sequence.status.seqActive;
   "Unit1.Em5.ControlNodes".mainPnP."step".action1[145] := #_w1 AND (NOT "Unit1.Em5.ControlNodes".cm.softCam.cathodeMainPnP1AxisZ.upPos.inPos OR NOT "Unit1.Em5.ControlNodes".cm.softCam.cathodeMainPnP2AxisZ.upPos.inPos);
   "Unit1.Em5.ControlNodes".mainPnP."step".transition1[145] := #_w1 AND "Unit1.Em5.ControlNodes".cm.softCam.cathodeMainPnP1AxisZ.upPos.inPos AND "Unit1.Em5.ControlNodes".cm.softCam.cathodeMainPnP2AxisZ.upPos.inPos;
   #statTonTime[145].TON(IN := #_w1 AND "Unit1.Em5.ControlNodes".mainPnP."step".transition1[145],
                         PT := #delayTime);
   IF #statTonTime[145].Q THEN
       "Unit1.Em5.ControlNodes".mainPnP.sequence.status.nextStep := #JOB_1_STEP_80;
   END_IF;
END_REGION

REGION Network 49: Step[180] : Main P&P 1,2 X-Axis Load Pos
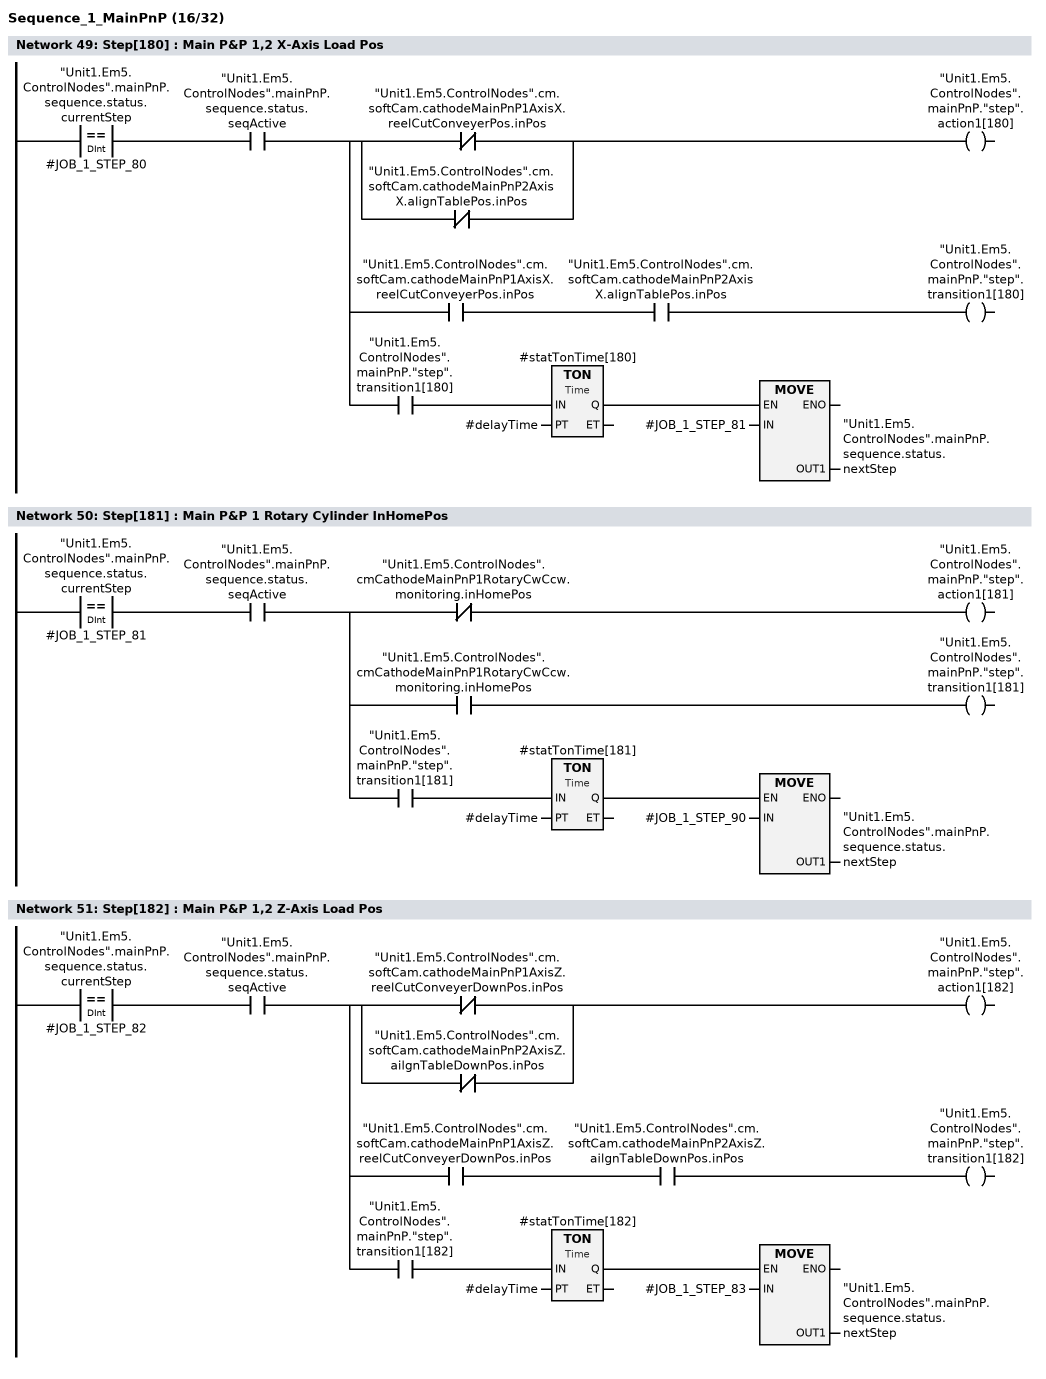
   RUNG wire#powerrail
      { S7_Templates := "SrcType := DInt" } EQ_Contact(in1 := "Unit1.Em5.ControlNodes".mainPnP.sequence.status.currentStep, in2 := #JOB_1_STEP_80)
      Contact( "Unit1.Em5.ControlNodes".mainPnP.sequence.status.seqActive )
      wire#w1
      I_Contact( "Unit1.Em5.ControlNodes".cm.softCam.cathodeMainPnP1AxisX.reelCutConveyerPos.inPos )
      wire#w2
      Coil( "Unit1.Em5.ControlNodes".mainPnP."step".action1[180] )
   END_RUNG
   RUNG wire#w1
      I_Contact( "Unit1.Em5.ControlNodes".cm.softCam.cathodeMainPnP2AxisX.alignTablePos.inPos )
   END_RUNG wire#w2
   RUNG wire#w1
      Contact( "Unit1.Em5.ControlNodes".cm.softCam.cathodeMainPnP1AxisX.reelCutConveyerPos.inPos )
      Contact( "Unit1.Em5.ControlNodes".cm.softCam.cathodeMainPnP2AxisX.alignTablePos.inPos )
      Coil( "Unit1.Em5.ControlNodes".mainPnP."step".transition1[180] )
   END_RUNG
   RUNG wire#w1
      Contact( "Unit1.Em5.ControlNodes".mainPnP."step".transition1[180] )
      { S7_Templates := "time_type := Time" } #statTonTime[180].TON(pt := #delayTime, et =>)
      Move(in := #JOB_1_STEP_81, out1 => "Unit1.Em5.ControlNodes".mainPnP.sequence.status.nextStep)
   END_RUNG
   // the same network as SCL:
   #_w1 := ("Unit1.Em5.ControlNodes".mainPnP.sequence.status.currentStep = #JOB_1_STEP_80) AND "Unit1.Em5.ControlNodes".mainPnP.sequence.status.seqActive;
   "Unit1.Em5.ControlNodes".mainPnP."step".action1[180] := #_w1 AND (NOT "Unit1.Em5.ControlNodes".cm.softCam.cathodeMainPnP1AxisX.reelCutConveyerPos.inPos OR NOT "Unit1.Em5.ControlNodes".cm.softCam.cathodeMainPnP2AxisX.alignTablePos.inPos);
   "Unit1.Em5.ControlNodes".mainPnP."step".transition1[180] := #_w1 AND "Unit1.Em5.ControlNodes".cm.softCam.cathodeMainPnP1AxisX.reelCutConveyerPos.inPos AND "Unit1.Em5.ControlNodes".cm.softCam.cathodeMainPnP2AxisX.alignTablePos.inPos;
   #statTonTime[180].TON(IN := #_w1 AND "Unit1.Em5.ControlNodes".mainPnP."step".transition1[180],
                         PT := #delayTime);
   IF #statTonTime[180].Q THEN
       "Unit1.Em5.ControlNodes".mainPnP.sequence.status.nextStep := #JOB_1_STEP_81;
   END_IF;
END_REGION

REGION Network 50: Step[181] : Main P&P 1 Rotary Cylinder InHomePos
   RUNG wire#powerrail
      { S7_Templates := "SrcType := DInt" } EQ_Contact(in1 := "Unit1.Em5.ControlNodes".mainPnP.sequence.status.currentStep, in2 := #JOB_1_STEP_81)
      Contact( "Unit1.Em5.ControlNodes".mainPnP.sequence.status.seqActive )
      wire#w1
      I_Contact( "Unit1.Em5.ControlNodes".cmCathodeMainPnP1RotaryCwCcw.monitoring.inHomePos )
      Coil( "Unit1.Em5.ControlNodes".mainPnP."step".action1[181] )
   END_RUNG
   RUNG wire#w1
      Contact( "Unit1.Em5.ControlNodes".cmCathodeMainPnP1RotaryCwCcw.monitoring.inHomePos )
      Coil( "Unit1.Em5.ControlNodes".mainPnP."step".transition1[181] )
   END_RUNG
   RUNG wire#w1
      Contact( "Unit1.Em5.ControlNodes".mainPnP."step".transition1[181] )
      { S7_Templates := "time_type := Time" } #statTonTime[181].TON(pt := #delayTime, et =>)
      Move(in := #JOB_1_STEP_90, out1 => "Unit1.Em5.ControlNodes".mainPnP.sequence.status.nextStep)
   END_RUNG
   // the same network as SCL:
   #_w1 := ("Unit1.Em5.ControlNodes".mainPnP.sequence.status.currentStep = #JOB_1_STEP_81) AND "Unit1.Em5.ControlNodes".mainPnP.sequence.status.seqActive;
   "Unit1.Em5.ControlNodes".mainPnP."step".action1[181] := #_w1 AND NOT "Unit1.Em5.ControlNodes".cmCathodeMainPnP1RotaryCwCcw.monitoring.inHomePos;
   "Unit1.Em5.ControlNodes".mainPnP."step".transition1[181] := #_w1 AND "Unit1.Em5.ControlNodes".cmCathodeMainPnP1RotaryCwCcw.monitoring.inHomePos;
   #statTonTime[181].TON(IN := #_w1 AND "Unit1.Em5.ControlNodes".mainPnP."step".transition1[181],
                         PT := #delayTime);
   IF #statTonTime[181].Q THEN
       "Unit1.Em5.ControlNodes".mainPnP.sequence.status.nextStep := #JOB_1_STEP_90;
   END_IF;
END_REGION

REGION Network 51: Step[182] : Main P&P 1,2 Z-Axis Load Pos
   RUNG wire#powerrail
      { S7_Templates := "SrcType := DInt" } EQ_Contact(in1 := "Unit1.Em5.ControlNodes".mainPnP.sequence.status.currentStep, in2 := #JOB_1_STEP_82)
      Contact( "Unit1.Em5.ControlNodes".mainPnP.sequence.status.seqActive )
      wire#w1
      I_Contact( "Unit1.Em5.ControlNodes".cm.softCam.cathodeMainPnP1AxisZ.reelCutConveyerDownPos.inPos )
      wire#w2
      Coil( "Unit1.Em5.ControlNodes".mainPnP."step".action1[182] )
   END_RUNG
   RUNG wire#w1
      I_Contact( "Unit1.Em5.ControlNodes".cm.softCam.cathodeMainPnP2AxisZ.ailgnTableDownPos.inPos )
   END_RUNG wire#w2
   RUNG wire#w1
      Contact( "Unit1.Em5.ControlNodes".cm.softCam.cathodeMainPnP1AxisZ.reelCutConveyerDownPos.inPos )
      Contact( "Unit1.Em5.ControlNodes".cm.softCam.cathodeMainPnP2AxisZ.ailgnTableDownPos.inPos )
      Coil( "Unit1.Em5.ControlNodes".mainPnP."step".transition1[182] )
   END_RUNG
   RUNG wire#w1
      Contact( "Unit1.Em5.ControlNodes".mainPnP."step".transition1[182] )
      { S7_Templates := "time_type := Time" } #statTonTime[182].TON(pt := #delayTime, et =>)
      Move(in := #JOB_1_STEP_83, out1 => "Unit1.Em5.ControlNodes".mainPnP.sequence.status.nextStep)
   END_RUNG
   // the same network as SCL:
   #_w1 := ("Unit1.Em5.ControlNodes".mainPnP.sequence.status.currentStep = #JOB_1_STEP_82) AND "Unit1.Em5.ControlNodes".mainPnP.sequence.status.seqActive;
   "Unit1.Em5.ControlNodes".mainPnP."step".action1[182] := #_w1 AND (NOT "Unit1.Em5.ControlNodes".cm.softCam.cathodeMainPnP1AxisZ.reelCutConveyerDownPos.inPos OR NOT "Unit1.Em5.ControlNodes".cm.softCam.cathodeMainPnP2AxisZ.ailgnTableDownPos.inPos);
   "Unit1.Em5.ControlNodes".mainPnP."step".transition1[182] := #_w1 AND "Unit1.Em5.ControlNodes".cm.softCam.cathodeMainPnP1AxisZ.reelCutConveyerDownPos.inPos AND "Unit1.Em5.ControlNodes".cm.softCam.cathodeMainPnP2AxisZ.ailgnTableDownPos.inPos;
   #statTonTime[182].TON(IN := #_w1 AND "Unit1.Em5.ControlNodes".mainPnP."step".transition1[182],
                         PT := #delayTime);
   IF #statTonTime[182].Q THEN
       "Unit1.Em5.ControlNodes".mainPnP.sequence.status.nextStep := #JOB_1_STEP_83;
   END_IF;
END_REGION

REGION Network 52: Step[183] : Main P&P 1,2 Vaccum On
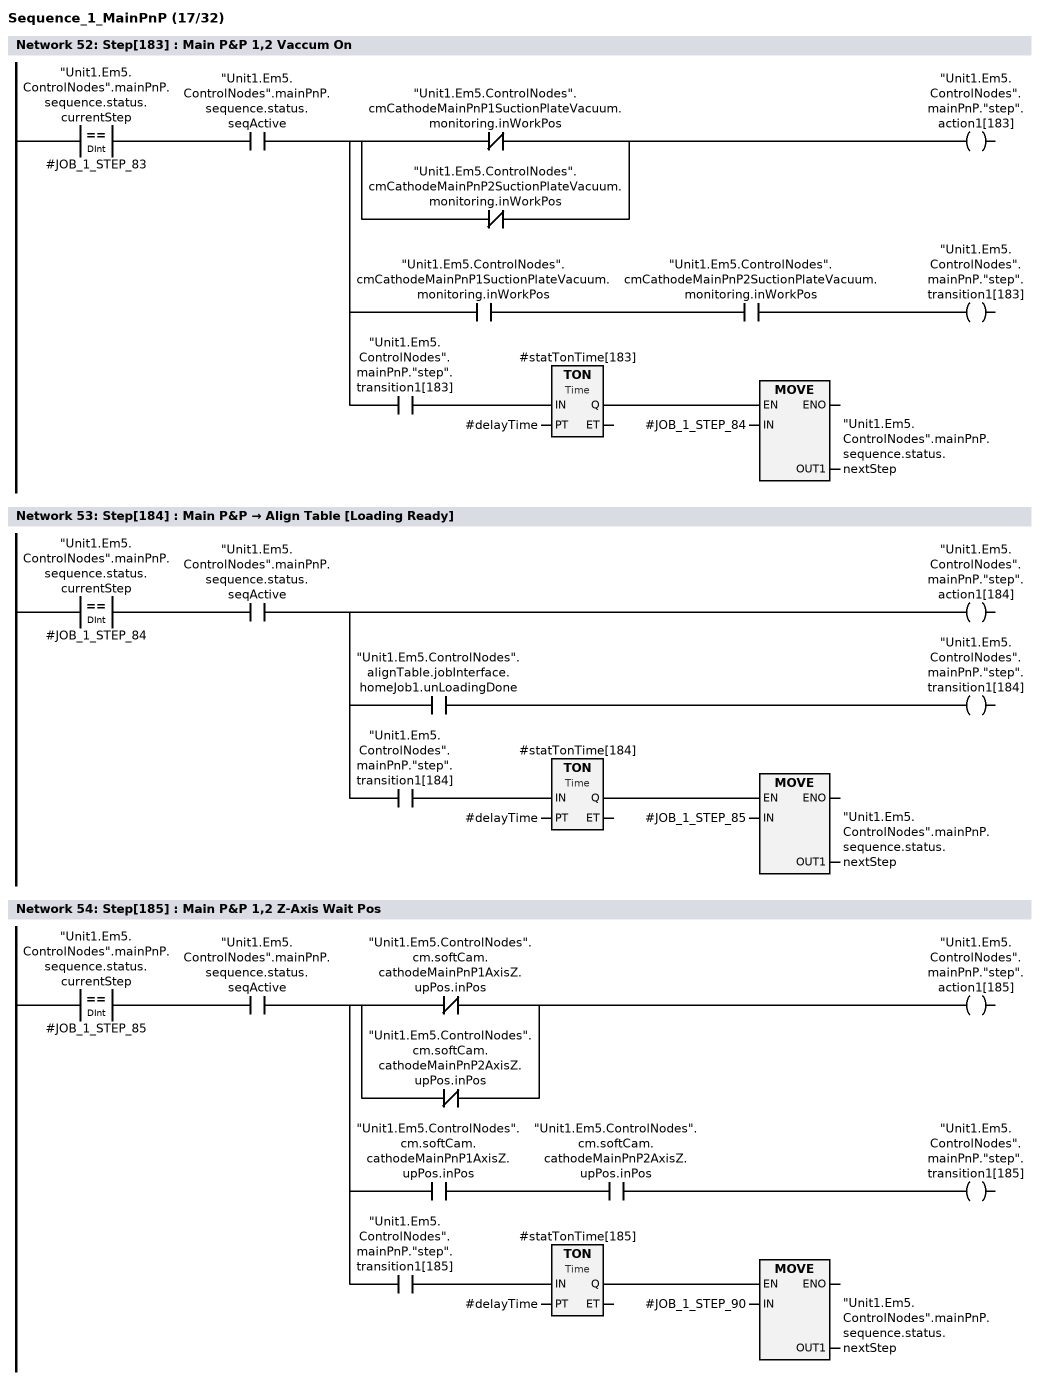
   RUNG wire#powerrail
      { S7_Templates := "SrcType := DInt" } EQ_Contact(in1 := "Unit1.Em5.ControlNodes".mainPnP.sequence.status.currentStep, in2 := #JOB_1_STEP_83)
      Contact( "Unit1.Em5.ControlNodes".mainPnP.sequence.status.seqActive )
      wire#w1
      I_Contact( "Unit1.Em5.ControlNodes".cmCathodeMainPnP1SuctionPlateVacuum.monitoring.inWorkPos )
      wire#w2
      Coil( "Unit1.Em5.ControlNodes".mainPnP."step".action1[183] )
   END_RUNG
   RUNG wire#w1
      I_Contact( "Unit1.Em5.ControlNodes".cmCathodeMainPnP2SuctionPlateVacuum.monitoring.inWorkPos )
   END_RUNG wire#w2
   RUNG wire#w1
      Contact( "Unit1.Em5.ControlNodes".cmCathodeMainPnP1SuctionPlateVacuum.monitoring.inWorkPos )
      Contact( "Unit1.Em5.ControlNodes".cmCathodeMainPnP2SuctionPlateVacuum.monitoring.inWorkPos )
      Coil( "Unit1.Em5.ControlNodes".mainPnP."step".transition1[183] )
   END_RUNG
   RUNG wire#w1
      Contact( "Unit1.Em5.ControlNodes".mainPnP."step".transition1[183] )
      { S7_Templates := "time_type := Time" } #statTonTime[183].TON(pt := #delayTime, et =>)
      Move(in := #JOB_1_STEP_84, out1 => "Unit1.Em5.ControlNodes".mainPnP.sequence.status.nextStep)
   END_RUNG
   // the same network as SCL:
   #_w1 := ("Unit1.Em5.ControlNodes".mainPnP.sequence.status.currentStep = #JOB_1_STEP_83) AND "Unit1.Em5.ControlNodes".mainPnP.sequence.status.seqActive;
   "Unit1.Em5.ControlNodes".mainPnP."step".action1[183] := #_w1 AND (NOT "Unit1.Em5.ControlNodes".cmCathodeMainPnP1SuctionPlateVacuum.monitoring.inWorkPos OR NOT "Unit1.Em5.ControlNodes".cmCathodeMainPnP2SuctionPlateVacuum.monitoring.inWorkPos);
   "Unit1.Em5.ControlNodes".mainPnP."step".transition1[183] := #_w1 AND "Unit1.Em5.ControlNodes".cmCathodeMainPnP1SuctionPlateVacuum.monitoring.inWorkPos AND "Unit1.Em5.ControlNodes".cmCathodeMainPnP2SuctionPlateVacuum.monitoring.inWorkPos;
   #statTonTime[183].TON(IN := #_w1 AND "Unit1.Em5.ControlNodes".mainPnP."step".transition1[183],
                         PT := #delayTime);
   IF #statTonTime[183].Q THEN
       "Unit1.Em5.ControlNodes".mainPnP.sequence.status.nextStep := #JOB_1_STEP_84;
   END_IF;
END_REGION

REGION Network 53: Step[184] : Main P&P → Align Table [Loading Ready]
   RUNG wire#powerrail
      { S7_Templates := "SrcType := DInt" } EQ_Contact(in1 := "Unit1.Em5.ControlNodes".mainPnP.sequence.status.currentStep, in2 := #JOB_1_STEP_84)
      Contact( "Unit1.Em5.ControlNodes".mainPnP.sequence.status.seqActive )
      wire#w1
      Coil( "Unit1.Em5.ControlNodes".mainPnP."step".action1[184] )
   END_RUNG
   RUNG wire#w1
      Contact( "Unit1.Em5.ControlNodes".alignTable.jobInterface.homeJob1.unLoadingDone )
      Coil( "Unit1.Em5.ControlNodes".mainPnP."step".transition1[184] )
   END_RUNG
   RUNG wire#w1
      Contact( "Unit1.Em5.ControlNodes".mainPnP."step".transition1[184] )
      { S7_Templates := "time_type := Time" } #statTonTime[184].TON(pt := #delayTime, et =>)
      Move(in := #JOB_1_STEP_85, out1 => "Unit1.Em5.ControlNodes".mainPnP.sequence.status.nextStep)
   END_RUNG
   // the same network as SCL:
   "Unit1.Em5.ControlNodes".mainPnP."step".action1[184] := ("Unit1.Em5.ControlNodes".mainPnP.sequence.status.currentStep = #JOB_1_STEP_84) AND "Unit1.Em5.ControlNodes".mainPnP.sequence.status.seqActive;
   "Unit1.Em5.ControlNodes".mainPnP."step".transition1[184] := ("Unit1.Em5.ControlNodes".mainPnP.sequence.status.currentStep = #JOB_1_STEP_84) AND "Unit1.Em5.ControlNodes".mainPnP.sequence.status.seqActive AND "Unit1.Em5.ControlNodes".alignTable.jobInterface.homeJob1.unLoadingDone;
   #statTonTime[184].TON(IN := ("Unit1.Em5.ControlNodes".mainPnP.sequence.status.currentStep = #JOB_1_STEP_84) AND "Unit1.Em5.ControlNodes".mainPnP.sequence.status.seqActive AND "Unit1.Em5.ControlNodes".mainPnP."step".transition1[184],
                         PT := #delayTime);
   IF #statTonTime[184].Q THEN
       "Unit1.Em5.ControlNodes".mainPnP.sequence.status.nextStep := #JOB_1_STEP_85;
   END_IF;
END_REGION

REGION Network 54: Step[185] : Main P&P 1,2 Z-Axis Wait Pos
   RUNG wire#powerrail
      { S7_Templates := "SrcType := DInt" } EQ_Contact(in1 := "Unit1.Em5.ControlNodes".mainPnP.sequence.status.currentStep, in2 := #JOB_1_STEP_85)
      Contact( "Unit1.Em5.ControlNodes".mainPnP.sequence.status.seqActive )
      wire#w1
      I_Contact( "Unit1.Em5.ControlNodes".cm.softCam.cathodeMainPnP1AxisZ.upPos.inPos )
      wire#w2
      Coil( "Unit1.Em5.ControlNodes".mainPnP."step".action1[185] )
   END_RUNG
   RUNG wire#w1
      I_Contact( "Unit1.Em5.ControlNodes".cm.softCam.cathodeMainPnP2AxisZ.upPos.inPos )
   END_RUNG wire#w2
   RUNG wire#w1
      Contact( "Unit1.Em5.ControlNodes".cm.softCam.cathodeMainPnP1AxisZ.upPos.inPos )
      Contact( "Unit1.Em5.ControlNodes".cm.softCam.cathodeMainPnP2AxisZ.upPos.inPos )
      Coil( "Unit1.Em5.ControlNodes".mainPnP."step".transition1[185] )
   END_RUNG
   RUNG wire#w1
      Contact( "Unit1.Em5.ControlNodes".mainPnP."step".transition1[185] )
      { S7_Templates := "time_type := Time" } #statTonTime[185].TON(pt := #delayTime, et =>)
      Move(in := #JOB_1_STEP_90, out1 => "Unit1.Em5.ControlNodes".mainPnP.sequence.status.nextStep)
   END_RUNG
   // the same network as SCL:
   #_w1 := ("Unit1.Em5.ControlNodes".mainPnP.sequence.status.currentStep = #JOB_1_STEP_85) AND "Unit1.Em5.ControlNodes".mainPnP.sequence.status.seqActive;
   "Unit1.Em5.ControlNodes".mainPnP."step".action1[185] := #_w1 AND (NOT "Unit1.Em5.ControlNodes".cm.softCam.cathodeMainPnP1AxisZ.upPos.inPos OR NOT "Unit1.Em5.ControlNodes".cm.softCam.cathodeMainPnP2AxisZ.upPos.inPos);
   "Unit1.Em5.ControlNodes".mainPnP."step".transition1[185] := #_w1 AND "Unit1.Em5.ControlNodes".cm.softCam.cathodeMainPnP1AxisZ.upPos.inPos AND "Unit1.Em5.ControlNodes".cm.softCam.cathodeMainPnP2AxisZ.upPos.inPos;
   #statTonTime[185].TON(IN := #_w1 AND "Unit1.Em5.ControlNodes".mainPnP."step".transition1[185],
                         PT := #delayTime);
   IF #statTonTime[185].Q THEN
       "Unit1.Em5.ControlNodes".mainPnP.sequence.status.nextStep := #JOB_1_STEP_90;
   END_IF;
END_REGION

REGION Network 55: Step[190] : JOB[1] Step End
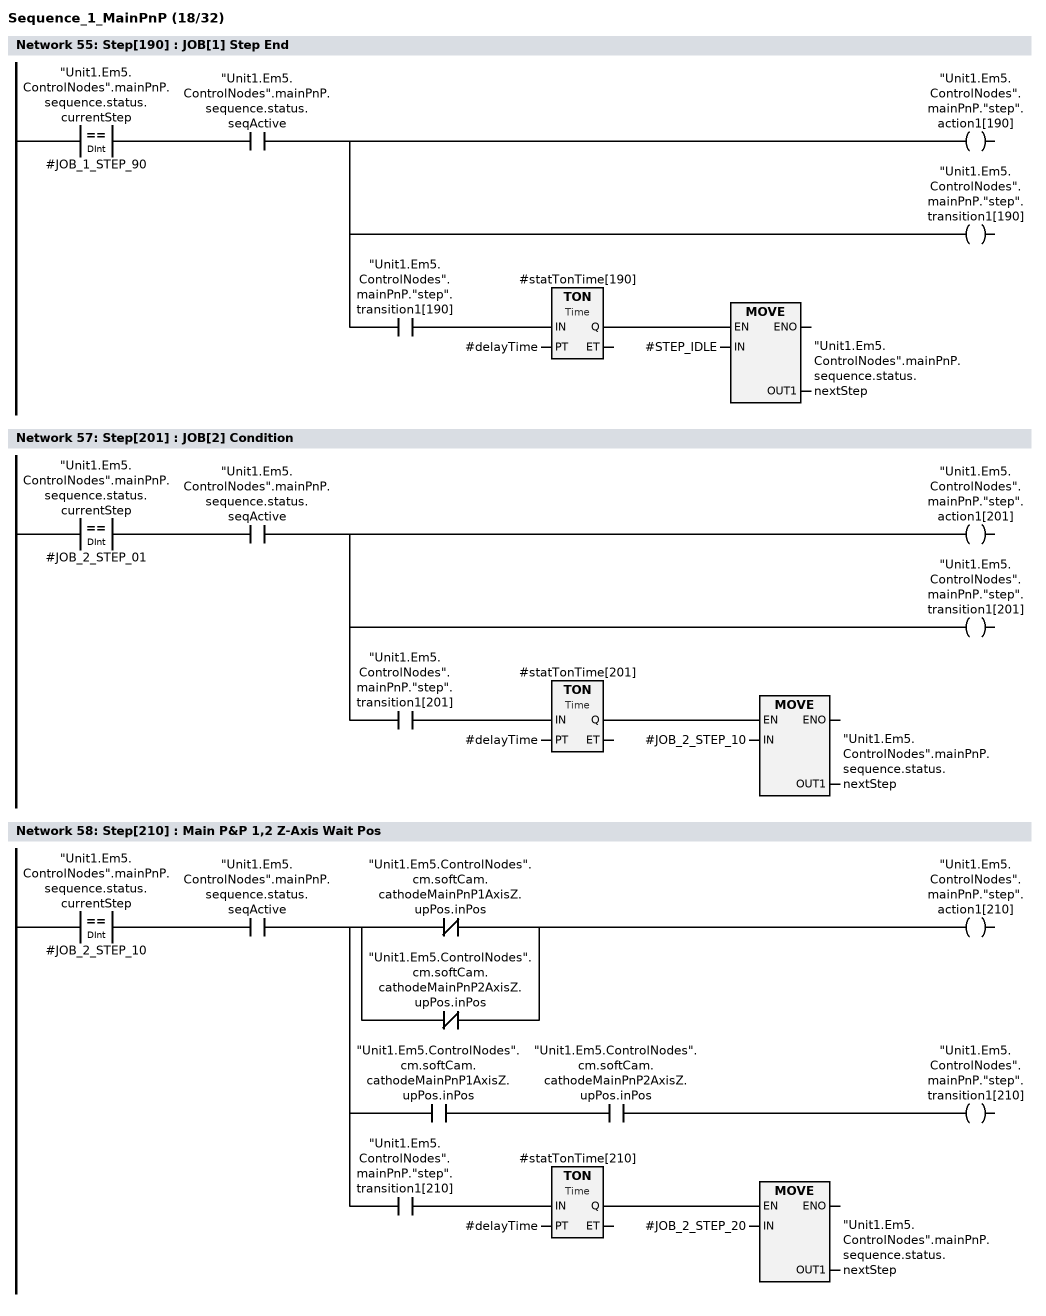
   RUNG wire#powerrail
      { S7_Templates := "SrcType := DInt" } EQ_Contact(in1 := "Unit1.Em5.ControlNodes".mainPnP.sequence.status.currentStep, in2 := #JOB_1_STEP_90)
      Contact( "Unit1.Em5.ControlNodes".mainPnP.sequence.status.seqActive )
      wire#w1
      Coil( "Unit1.Em5.ControlNodes".mainPnP."step".action1[190] )
   END_RUNG
   RUNG wire#w1
      Coil( "Unit1.Em5.ControlNodes".mainPnP."step".transition1[190] )
   END_RUNG
   RUNG wire#w1
      Contact( "Unit1.Em5.ControlNodes".mainPnP."step".transition1[190] )
      { S7_Templates := "time_type := Time" } #statTonTime[190].TON(pt := #delayTime, et =>)
      Move(in := #STEP_IDLE, out1 => "Unit1.Em5.ControlNodes".mainPnP.sequence.status.nextStep)
   END_RUNG
   // the same network as SCL:
   "Unit1.Em5.ControlNodes".mainPnP."step".action1[190] := ("Unit1.Em5.ControlNodes".mainPnP.sequence.status.currentStep = #JOB_1_STEP_90) AND "Unit1.Em5.ControlNodes".mainPnP.sequence.status.seqActive;
   "Unit1.Em5.ControlNodes".mainPnP."step".transition1[190] := ("Unit1.Em5.ControlNodes".mainPnP.sequence.status.currentStep = #JOB_1_STEP_90) AND "Unit1.Em5.ControlNodes".mainPnP.sequence.status.seqActive;
   #statTonTime[190].TON(IN := ("Unit1.Em5.ControlNodes".mainPnP.sequence.status.currentStep = #JOB_1_STEP_90) AND "Unit1.Em5.ControlNodes".mainPnP.sequence.status.seqActive AND "Unit1.Em5.ControlNodes".mainPnP."step".transition1[190],
                         PT := #delayTime);
   IF #statTonTime[190].Q THEN
       "Unit1.Em5.ControlNodes".mainPnP.sequence.status.nextStep := #STEP_IDLE;
   END_IF;
END_REGION

REGION Network 56: *************** JOB[2] Loading ************************
END_REGION

REGION Network 57: Step[201] : JOB[2] Condition
   RUNG wire#powerrail
      { S7_Templates := "SrcType := DInt" } EQ_Contact(in1 := "Unit1.Em5.ControlNodes".mainPnP.sequence.status.currentStep, in2 := #JOB_2_STEP_01)
      Contact( "Unit1.Em5.ControlNodes".mainPnP.sequence.status.seqActive )
      wire#w1
      Coil( "Unit1.Em5.ControlNodes".mainPnP."step".action1[201] )
   END_RUNG
   RUNG wire#w1
      Coil( "Unit1.Em5.ControlNodes".mainPnP."step".transition1[201] )
   END_RUNG
   RUNG wire#w1
      Contact( "Unit1.Em5.ControlNodes".mainPnP."step".transition1[201] )
      { S7_Templates := "time_type := Time" } #statTonTime[201].TON(pt := #delayTime, et =>)
      Move(in := #JOB_2_STEP_10, out1 => "Unit1.Em5.ControlNodes".mainPnP.sequence.status.nextStep)
   END_RUNG
   // the same network as SCL:
   "Unit1.Em5.ControlNodes".mainPnP."step".action1[201] := ("Unit1.Em5.ControlNodes".mainPnP.sequence.status.currentStep = #JOB_2_STEP_01) AND "Unit1.Em5.ControlNodes".mainPnP.sequence.status.seqActive;
   "Unit1.Em5.ControlNodes".mainPnP."step".transition1[201] := ("Unit1.Em5.ControlNodes".mainPnP.sequence.status.currentStep = #JOB_2_STEP_01) AND "Unit1.Em5.ControlNodes".mainPnP.sequence.status.seqActive;
   #statTonTime[201].TON(IN := ("Unit1.Em5.ControlNodes".mainPnP.sequence.status.currentStep = #JOB_2_STEP_01) AND "Unit1.Em5.ControlNodes".mainPnP.sequence.status.seqActive AND "Unit1.Em5.ControlNodes".mainPnP."step".transition1[201],
                         PT := #delayTime);
   IF #statTonTime[201].Q THEN
       "Unit1.Em5.ControlNodes".mainPnP.sequence.status.nextStep := #JOB_2_STEP_10;
   END_IF;
END_REGION

